C09080=1062.596,-86.701,-61.931,171.565,25.593,154.776
C09081=1062.602,-86.451,-61.943,171.566,25.594,154.776
C09082=1062.608,-86.202,-61.953,171.568,25.596,154.777
C09083=1062.614,-85.953,-61.964,171.570,25.597,154.777
C09084=1062.620,-85.702,-61.975,171.571,25.598,154.777
C09085=1062.627,-85.453,-61.985,171.573,25.600,154.777
C09086=1062.633,-85.204,-61.996,171.575,25.601,154.777
C09087=1062.639,-84.954,-62.007,171.576,25.603,154.777
C09088=1062.646,-84.704,-62.018,171.578,25.604,154.777
C09089=1062.652,-84.454,-62.028,171.580,25.605,154.777
C09090=1062.657,-84.204,-62.039,171.581,25.607,154.777
C09091=1062.664,-83.955,-62.049,171.583,25.608,154.777
C09092=1062.670,-83.705,-62.061,171.585,25.609,154.777
C09093=1062.676,-83.455,-62.072,171.587,25.611,154.777
C09094=1062.682,-83.206,-62.082,171.589,25.613,154.777
C09095=1062.689,-82.956,-62.093,171.591,25.614,154.777
C09096=1062.696,-82.674,-62.105,171.592,25.616,154.777
C09097=1062.703,-82.392,-62.118,171.594,25.617,154.778
C09098=1062.709,-82.110,-62.130,171.597,25.619,154.778
C09099=1062.716,-81.829,-62.143,171.598,25.621,154.778
C09100=1062.723,-81.579,-62.154,171.600,25.622,154.778
C09101=1062.729,-81.329,-62.164,171.602,25.624,154.778
C09102=1062.736,-81.079,-62.176,171.603,25.625,154.778
C09103=1062.741,-80.830,-62.187,171.605,25.627,154.778
C09104=1062.748,-80.580,-62.197,171.607,25.628,154.778
C09105=1062.754,-80.330,-62.208,171.608,25.630,154.778
C09106=1062.760,-80.081,-62.219,171.610,25.631,154.778
C09107=1062.766,-79.831,-62.230,171.612,25.632,154.778
C09108=1062.773,-79.582,-62.240,171.613,25.634,154.778
C09109=1062.779,-79.331,-62.252,171.615,25.635,154.778
C09110=1062.785,-79.082,-62.263,171.617,25.637,154.778
C09111=1062.791,-78.832,-62.274,171.619,25.639,154.779
C09112=1062.797,-78.583,-62.285,171.621,25.640,154.779
C09113=1062.803,-78.333,-62.296,171.622,25.642,154.779
C09114=1062.809,-78.083,-62.308,171.624,25.644,154.779
C09115=1062.815,-77.834,-62.318,171.626,25.645,154.779
C09116=1062.821,-77.583,-62.330,171.627,25.646,154.779
C09117=1062.827,-77.334,-62.341,171.629,25.648,154.779
C09118=1062.834,-77.084,-62.353,171.631,25.649,154.779
C09119=1062.839,-76.835,-62.363,171.632,25.651,154.779
C09120=1062.846,-76.585,-62.375,171.634,25.652,154.779
C09121=1062.851,-76.335,-62.386,171.636,25.654,154.779
C09122=1062.857,-76.086,-62.396,171.637,25.656,154.780
C09123=1062.864,-75.836,-62.408,171.639,25.657,154.780
C09124=1062.870,-75.587,-62.419,171.640,25.659,154.780
C09125=1062.877,-75.337,-62.430,171.642,25.661,154.780
C09126=1062.882,-75.087,-62.441,171.644,25.662,154.780
C09127=1062.889,-74.838,-62.453,171.645,25.664,154.780
C09128=1062.895,-74.588,-62.464,171.647,25.665,154.780
C09129=1062.901,-74.338,-62.475,171.650,25.667,154.780
C09130=1062.907,-74.089,-62.486,171.651,25.669,154.780
C09131=1062.914,-73.839,-62.498,171.653,25.671,154.780
C09132=1062.919,-73.589,-62.509,171.654,25.672,154.781
C09133=1062.925,-73.339,-62.520,171.656,25.673,154.781
C09134=1062.931,-73.090,-62.532,171.658,25.675,154.781
C09135=1062.937,-72.840,-62.543,171.659,25.677,154.781
C09136=1062.943,-72.590,-62.554,171.661,25.679,154.781
C09137=1062.950,-72.341,-62.566,171.663,25.681,154.781
C09138=1062.955,-72.091,-62.578,171.664,25.682,154.781
C09139=1062.960,-71.842,-62.588,171.666,25.684,154.781
C09140=1062.967,-71.592,-62.600,171.668,25.685,154.782
C09141=1062.973,-71.342,-62.611,171.669,25.687,154.782
C09142=1062.979,-71.092,-62.622,171.671,25.689,154.782
C09143=1062.984,-70.843,-62.635,171.672,25.691,154.782
C09144=1062.991,-70.593,-62.646,171.674,25.692,154.782
C09145=1062.997,-70.344,-62.658,171.676,25.694,154.782
C09146=1063.003,-70.094,-62.669,171.677,25.696,154.782
C09147=1063.008,-69.844,-62.680,171.679,25.698,154.783
C09148=1063.015,-69.594,-62.692,171.680,25.699,154.783
C09149=1063.021,-69.345,-62.703,171.682,25.701,154.783
C09150=1063.027,-69.095,-62.715,171.684,25.702,154.783
C09151=1063.034,-68.845,-62.726,171.686,25.705,154.783
C09152=1063.039,-68.596,-62.738,171.688,25.706,154.783
C09153=1063.045,-68.346,-62.750,171.689,25.708,154.783
C09154=1063.051,-68.096,-62.761,171.691,25.710,154.783
C09155=1063.058,-67.847,-62.773,171.693,25.712,154.783
C09156=1063.063,-67.597,-62.784,171.694,25.713,154.784
C09157=1063.069,-67.347,-62.796,171.696,25.715,154.784
C09158=1063.075,-67.098,-62.807,171.697,25.717,154.784
C09159=1063.082,-66.848,-62.819,171.699,25.719,154.784
C09160=1063.088,-66.569,-62.832,171.701,25.721,154.784
C09161=1063.095,-66.289,-62.845,171.702,25.722,154.784
C09162=1063.102,-66.009,-62.858,171.705,25.724,154.784
C09163=1063.108,-65.729,-62.871,171.706,25.726,154.785
C09164=1063.114,-65.480,-62.883,171.708,25.728,154.785
C09165=1063.121,-65.230,-62.895,171.710,25.730,154.785
C09166=1063.127,-64.981,-62.906,171.711,25.731,154.785
C09167=1063.132,-64.731,-62.918,171.713,25.733,154.785
C09168=1063.139,-64.481,-62.929,171.714,25.735,154.785
C09169=1063.145,-64.232,-62.941,171.716,25.737,154.785
C09170=1063.151,-63.982,-62.952,171.718,25.739,154.786
C09171=1063.157,-63.732,-62.965,171.719,25.740,154.786
C09172=1063.163,-63.483,-62.976,171.721,25.742,154.786
C09173=1063.169,-63.233,-62.988,171.723,25.744,154.786
C09174=1063.175,-62.984,-63.000,171.725,25.746,154.786
C09175=1063.181,-62.733,-63.011,171.726,25.748,154.786
C09176=1063.188,-62.484,-63.023,171.728,25.749,154.786
C09177=1063.194,-62.235,-63.035,171.730,25.751,154.786
C09178=1063.199,-61.984,-63.046,171.731,25.754,154.787
C09179=1063.206,-61.735,-63.058,171.733,25.755,154.787
C09180=1063.212,-61.486,-63.070,171.734,25.757,154.787
C09181=1063.218,-61.235,-63.082,171.736,25.759,154.787
C09182=1063.224,-60.986,-63.094,171.738,25.761,154.787
C09183=1063.230,-60.737,-63.105,171.739,25.762,154.787
C09184=1063.236,-60.486,-63.117,171.741,25.764,154.788
C09185=1063.243,-60.237,-63.129,171.742,25.766,154.788
C09186=1063.249,-59.987,-63.141,171.744,25.768,154.788
C09187=1063.255,-59.738,-63.153,171.746,25.769,154.788
C09188=1063.261,-59.488,-63.164,171.747,25.771,154.788
C09189=1063.268,-59.238,-63.176,171.749,25.773,154.788
C09190=1063.273,-58.989,-63.189,171.750,25.775,154.788
C09191=1063.280,-58.740,-63.201,171.752,25.777,154.789
C09192=1063.286,-58.489,-63.212,171.754,25.778,154.789
C09193=1063.292,-58.240,-63.224,171.755,25.780,154.789
C09194=1063.298,-57.991,-63.236,171.757,25.782,154.789
C09195=1063.304,-57.741,-63.248,171.758,25.784,154.789
C09196=1063.310,-57.491,-63.260,171.760,25.786,154.789
C09197=1063.317,-57.241,-63.272,171.762,25.788,154.790
C09198=1063.323,-56.992,-63.283,171.764,25.790,154.790
C09199=1063.329,-56.742,-63.296,171.766,25.792,154.790
C09200=1063.335,-56.493,-63.308,171.767,25.793,154.790
C09201=1063.342,-56.243,-63.319,171.769,25.795,154.790
C09202=1063.347,-55.993,-63.331,171.770,25.797,154.790
C09203=1063.354,-55.744,-63.343,171.772,25.799,154.791
C09204=1063.360,-55.494,-63.355,171.774,25.801,154.791
C09205=1063.366,-55.244,-63.368,171.775,25.803,154.791
C09206=1063.373,-54.995,-63.380,171.777,25.805,154.791
C09207=1063.378,-54.746,-63.392,171.778,25.806,154.791
C09208=1063.384,-54.495,-63.403,171.780,25.808,154.791
C09209=1063.391,-54.246,-63.415,171.781,25.810,154.791
C09210=1063.397,-53.996,-63.428,171.783,25.812,154.792
C09211=1063.404,-53.746,-63.440,171.785,25.814,154.792
C09212=1063.409,-53.497,-63.452,171.786,25.816,154.792
C09213=1063.416,-53.248,-63.464,171.788,25.817,154.792
C09214=1063.422,-52.998,-63.476,171.790,25.819,154.792
C09215=1063.428,-52.748,-63.488,171.791,25.822,154.792
C09216=1063.435,-52.499,-63.500,171.793,25.823,154.793
C09217=1063.441,-52.249,-63.513,171.794,25.825,154.793
C09218=1063.447,-51.999,-63.525,171.796,25.827,154.793
C09219=1063.453,-51.750,-63.536,171.797,25.829,154.793
C09220=1063.459,-51.500,-63.549,171.799,25.830,154.793
C09221=1063.466,-51.250,-63.560,171.801,25.833,154.793
C09222=1063.472,-51.000,-63.573,171.803,25.835,154.794
C09223=1063.478,-50.751,-63.585,171.805,25.837,154.794
C09224=1063.485,-50.473,-63.599,171.806,25.839,154.794
C09225=1063.492,-50.195,-63.612,171.808,25.841,154.794
C09226=1063.499,-49.916,-63.626,171.809,25.843,154.794
C09227=1063.506,-49.637,-63.640,171.812,25.845,154.794
C09228=1063.511,-49.387,-63.652,171.813,25.847,154.795
C09229=1063.518,-49.138,-63.664,171.815,25.849,154.795
C09230=1063.523,-48.889,-63.676,171.816,25.852,154.795
C09231=1063.529,-48.639,-63.689,171.818,25.853,154.795
C09232=1063.535,-48.389,-63.701,171.820,25.855,154.795
C09233=1063.542,-48.140,-63.714,171.821,25.857,154.796
C09234=1063.548,-47.890,-63.727,171.823,25.859,154.796
C09235=1063.554,-47.640,-63.739,171.824,25.862,154.796
C09236=1063.560,-47.391,-63.751,171.826,25.863,154.796
C09237=1063.566,-47.141,-63.763,171.827,25.866,154.796
C09238=1063.572,-46.891,-63.776,171.829,25.867,154.797
C09239=1063.578,-46.642,-63.788,171.830,25.870,154.797
C09240=1063.584,-46.392,-63.800,171.832,25.872,154.797
C09241=1063.591,-46.143,-63.814,171.834,25.873,154.797
C09242=1063.597,-45.893,-63.826,171.835,25.876,154.797
C09243=1063.602,-45.644,-63.838,171.837,25.877,154.798
C09244=1063.609,-45.394,-63.850,171.838,25.880,154.798
C09245=1063.614,-45.144,-63.863,171.840,25.881,154.798
C09246=1063.620,-44.894,-63.875,171.841,25.884,154.798
C09247=1063.627,-44.645,-63.888,171.843,25.886,154.798
C09248=1063.633,-44.396,-63.901,171.844,25.888,154.799
C09249=1063.639,-44.146,-63.913,171.846,25.890,154.799
C09250=1063.645,-43.896,-63.926,171.847,25.892,154.799
C09251=1063.652,-43.646,-63.938,171.849,25.894,154.799
C09252=1063.657,-43.398,-63.951,171.851,25.896,154.799
C09253=1063.663,-43.148,-63.963,171.852,25.898,154.800
C09254=1063.669,-42.898,-63.976,171.854,25.900,154.800
C09255=1063.675,-42.648,-63.988,171.855,25.902,154.800
C09256=1063.682,-42.399,-64.001,171.857,25.904,154.800
C09257=1063.688,-42.149,-64.013,171.858,25.906,154.800
C09258=1063.694,-41.899,-64.026,171.860,25.908,154.801
C09259=1063.700,-41.649,-64.039,171.862,25.910,154.801
C09260=1063.707,-41.400,-64.051,171.864,25.912,154.801
C09261=1063.713,-41.151,-64.064,171.865,25.915,154.801
C09262=1063.718,-40.901,-64.076,171.867,25.917,154.801
C09263=1063.725,-40.651,-64.090,171.869,25.919,154.802
C09264=1063.731,-40.402,-64.102,171.870,25.921,154.802
C09265=1063.737,-40.152,-64.114,171.872,25.923,154.802
C09266=1063.743,-39.903,-64.127,171.873,25.925,154.802
C09267=1063.749,-39.653,-64.140,171.875,25.927,154.802
C09268=1063.755,-39.403,-64.153,171.876,25.929,154.803
C09269=1063.761,-39.154,-64.166,171.878,25.931,154.803
C09270=1063.768,-38.904,-64.178,171.879,25.933,154.803
C09271=1063.774,-38.654,-64.190,171.881,25.935,154.803
C09272=1063.780,-38.405,-64.204,171.882,25.937,154.804
C09273=1063.786,-38.155,-64.216,171.884,25.940,154.804
C09274=1063.792,-37.906,-64.229,171.886,25.941,154.804
C09275=1063.798,-37.656,-64.242,171.887,25.944,154.804
C09276=1063.804,-37.406,-64.255,171.889,25.946,154.804
C09277=1063.810,-37.157,-64.268,171.890,25.948,154.805
C09278=1063.816,-36.907,-64.280,171.892,25.950,154.805
C09279=1063.823,-36.658,-64.294,171.893,25.953,154.805
C09280=1063.828,-36.408,-64.306,171.895,25.954,154.805
C09281=1063.835,-36.158,-64.319,171.896,25.957,154.806
C09282=1063.841,-35.909,-64.332,171.898,25.959,154.806
C09283=1063.847,-35.659,-64.345,171.899,25.961,154.806
C09284=1063.853,-35.409,-64.358,171.901,25.963,154.806
C09285=1063.859,-35.160,-64.371,171.902,25.965,154.807
C09286=1063.865,-34.910,-64.384,171.904,25.967,154.807
C09287=1063.871,-34.661,-64.397,171.905,25.970,154.807
C09288=1063.877,-34.382,-64.411,171.907,25.972,154.807
C09289=1063.884,-34.105,-64.425,171.908,25.974,154.807
C09290=1063.891,-33.827,-64.439,171.911,25.977,154.808
C09291=1063.897,-33.548,-64.454,171.912,25.979,154.808
C09292=1063.904,-33.299,-64.468,171.914,25.981,154.808
C09293=1063.910,-33.049,-64.480,171.915,25.984,154.808
C09294=1063.916,-32.800,-64.494,171.917,25.986,154.809
C09295=1063.922,-32.551,-64.507,171.918,25.988,154.809
C09296=1063.928,-32.301,-64.519,171.920,25.990,154.809
C09297=1063.934,-32.051,-64.533,171.921,25.993,154.809
C09298=1063.940,-31.801,-64.545,171.923,25.994,154.810
C09299=1063.946,-31.552,-64.558,171.924,25.997,154.810
C09300=1063.952,-31.303,-64.572,171.926,25.999,154.810
C09301=1063.958,-31.053,-64.584,171.927,26.001,154.810
C09302=1063.965,-30.804,-64.598,171.929,26.003,154.811
C09303=1063.971,-30.554,-64.610,171.931,26.005,154.811
C09304=1063.977,-30.304,-64.624,171.932,26.008,154.811
C09305=1063.984,-30.055,-64.637,171.934,26.010,154.811
C09306=1063.989,-29.805,-64.650,171.935,26.012,154.811
C09307=1063.995,-29.555,-64.663,171.937,26.014,154.812
C09308=1064.001,-29.306,-64.677,171.938,26.016,154.812
C09309=1064.007,-29.056,-64.689,171.940,26.019,154.812
C09310=1064.013,-28.807,-64.702,171.941,26.021,154.812
C09311=1064.019,-28.558,-64.716,171.943,26.023,154.813
C09312=1064.026,-28.307,-64.729,171.944,26.025,154.813
C09313=1064.032,-28.058,-64.742,171.946,26.028,154.813
C09314=1064.038,-27.808,-64.755,171.947,26.029,154.813
C09315=1064.045,-27.559,-64.768,171.949,26.032,154.814
C09316=1064.051,-27.309,-64.781,171.950,26.034,154.814
C09317=1064.056,-27.060,-64.795,171.952,26.036,154.814
C09318=1064.063,-26.810,-64.809,171.953,26.039,154.814
C09319=1064.069,-26.561,-64.822,171.955,26.040,154.815
C09320=1064.075,-26.311,-64.834,171.956,26.043,154.815
C09321=1064.080,-26.061,-64.848,171.958,26.045,154.815
C09322=1064.087,-25.812,-64.861,171.959,26.047,154.815
C09323=1064.093,-25.563,-64.875,171.961,26.050,154.816
C09324=1064.099,-25.313,-64.887,171.962,26.052,154.816
C09325=1064.104,-25.063,-64.901,171.964,26.054,154.816
C09326=1064.111,-24.813,-64.915,171.965,26.057,154.816
C09327=1064.117,-24.564,-64.928,171.967,26.059,154.817
C09328=1064.123,-24.314,-64.942,171.968,26.061,154.817
C09329=1064.129,-24.065,-64.955,171.970,26.064,154.817
C09330=1064.135,-23.815,-64.968,171.971,26.066,154.817
C09331=1064.140,-23.566,-64.982,171.973,26.068,154.818
C09332=1064.147,-23.316,-64.995,171.975,26.070,154.818
C09333=1064.153,-23.066,-65.009,171.976,26.072,154.818
C09334=1064.159,-22.817,-65.022,171.978,26.075,154.818
C09335=1064.165,-22.567,-65.036,171.979,26.077,154.819
C09336=1064.171,-22.318,-65.049,171.981,26.079,154.819
C09337=1064.177,-22.069,-65.063,171.982,26.082,154.819
C09338=1064.183,-21.818,-65.076,171.984,26.084,154.820
C09339=1064.189,-21.569,-65.089,171.985,26.086,154.820
C09340=1064.195,-21.319,-65.103,171.987,26.089,154.820
C09341=1064.201,-21.070,-65.116,171.988,26.091,154.820
C09342=1064.207,-20.821,-65.129,171.990,26.093,154.821
C09343=1064.213,-20.570,-65.144,171.991,26.096,154.821
C09344=1064.220,-20.321,-65.157,171.993,26.098,154.821
C09345=1064.226,-20.072,-65.170,171.994,26.100,154.821
C09346=1064.231,-19.822,-65.184,171.996,26.103,154.822
C09347=1064.238,-19.572,-65.198,171.997,26.105,154.822
C09348=1064.244,-19.323,-65.211,171.999,26.107,154.822
C09349=1064.250,-19.074,-65.225,172.000,26.110,154.822
C09350=1064.256,-18.824,-65.238,172.002,26.112,154.823
C09351=1064.263,-18.574,-65.252,172.003,26.114,154.823
C09352=1064.269,-18.295,-65.267,172.005,26.117,154.823
C09353=1064.276,-18.016,-65.283,172.006,26.119,154.824
C09354=1064.282,-17.738,-65.298,172.008,26.122,154.824
C09355=1064.289,-17.459,-65.313,172.010,26.124,154.824
C09356=1064.295,-17.210,-65.326,172.011,26.127,154.824
C09357=1064.302,-16.960,-65.340,172.013,26.129,154.825
C09358=1064.308,-16.710,-65.354,172.014,26.131,154.825
C09359=1064.314,-16.461,-65.367,172.016,26.134,154.825
C09360=1064.320,-16.211,-65.381,172.017,26.136,154.825
C09361=1064.326,-15.961,-65.394,172.019,26.138,154.826
C09362=1064.333,-15.713,-65.408,172.020,26.141,154.826
C09363=1064.338,-15.463,-65.422,172.022,26.143,154.826
C09364=1064.345,-15.213,-65.436,172.023,26.145,154.827
C09365=1064.351,-14.964,-65.450,172.025,26.148,154.827
C09366=1064.357,-14.714,-65.463,172.026,26.150,154.827
C09367=1064.363,-14.464,-65.477,172.028,26.152,154.827
C09368=1064.369,-14.215,-65.490,172.029,26.155,154.828
C09369=1064.375,-13.965,-65.504,172.031,26.157,154.828
C09370=1064.380,-13.716,-65.519,172.032,26.159,154.828
C09371=1064.387,-13.466,-65.533,172.034,26.162,154.829
C09372=1064.393,-13.217,-65.546,172.035,26.164,154.829
C09373=1064.399,-12.967,-65.560,172.037,26.167,154.829
C09374=1064.405,-12.717,-65.574,172.038,26.169,154.829
C09375=1064.411,-12.468,-65.588,172.040,26.171,154.830
C09376=1064.417,-12.219,-65.602,172.041,26.174,154.830
C09377=1064.423,-11.969,-65.616,172.043,26.176,154.830
C09378=1064.429,-11.719,-65.629,172.043,26.178,154.830
C09379=1064.435,-11.470,-65.643,172.045,26.181,154.831
C09380=1064.441,-11.220,-65.658,172.046,26.183,154.831
C09381=1064.447,-10.971,-65.671,172.048,26.186,154.831
C09382=1064.453,-10.721,-65.685,172.049,26.188,154.832
C09383=1064.459,-10.471,-65.699,172.051,26.190,154.832
C09384=1064.465,-10.222,-65.713,172.052,26.192,154.832
C09385=1064.471,-9.973,-65.727,172.054,26.195,154.832
C09386=1064.478,-9.723,-65.741,172.055,26.198,154.833
C09387=1064.483,-9.474,-65.756,172.057,26.200,154.833
C09388=1064.489,-9.224,-65.769,172.058,26.202,154.833
C09389=1064.496,-8.974,-65.783,172.060,26.205,154.834
C09390=1064.501,-8.725,-65.798,172.061,26.207,154.834
C09391=1064.508,-8.475,-65.812,172.063,26.209,154.834
C09392=1064.514,-8.226,-65.825,172.064,26.212,154.835
C09393=1064.520,-7.977,-65.840,172.066,26.214,154.835
C09394=1064.526,-7.727,-65.854,172.067,26.217,154.835
C09395=1064.532,-7.477,-65.867,172.069,26.219,154.835
C09396=1064.538,-7.228,-65.882,172.070,26.221,154.836
C09397=1064.544,-6.978,-65.896,172.072,26.224,154.836
C09398=1064.550,-6.729,-65.909,172.073,26.227,154.836
C09399=1064.556,-6.479,-65.924,172.075,26.229,154.837
C09400=1064.562,-6.230,-65.938,172.076,26.231,154.837
C09401=1064.569,-5.980,-65.952,172.078,26.234,154.837
C09402=1064.574,-5.731,-65.966,172.079,26.236,154.837
C09403=1064.580,-5.480,-65.980,172.081,26.238,154.838
C09404=1064.587,-5.232,-65.994,172.082,26.241,154.838
C09405=1064.592,-4.982,-66.008,172.084,26.243,154.838
C09406=1064.599,-4.733,-66.023,172.085,26.246,154.839
C09407=1064.605,-4.483,-66.037,172.087,26.248,154.839
C09408=1064.611,-4.234,-66.052,172.088,26.250,154.839
C09409=1064.617,-3.984,-66.065,172.090,26.253,154.839
C09410=1064.623,-3.734,-66.080,172.091,26.256,154.840
C09411=1064.630,-3.485,-66.094,172.092,26.258,154.840
C09412=1064.636,-3.235,-66.108,172.094,26.260,154.840
C09413=1064.641,-2.986,-66.122,172.095,26.262,154.841
C09414=1064.647,-2.736,-66.137,172.097,26.265,154.841
C09415=1064.653,-2.487,-66.151,172.097,26.267,154.841
C09416=1064.660,-2.206,-66.168,172.100,26.271,154.842
C09417=1064.667,-1.926,-66.183,172.101,26.273,154.842
C09418=1064.674,-1.645,-66.199,172.103,26.276,154.842
C09419=1064.680,-1.365,-66.216,172.104,26.279,154.843
C09420=1064.685,-1.116,-66.230,172.106,26.281,154.843
C09421=1064.692,-0.866,-66.245,172.107,26.284,154.843
C09422=1064.697,-0.616,-66.259,172.108,26.286,154.844
C09423=1064.704,-0.367,-66.274,172.110,26.288,154.844
C09424=1064.709,-0.117,-66.288,172.111,26.291,154.844
C09425=1064.716,0.132,-66.302,172.113,26.294,154.845
C09426=1064.722,0.381,-66.317,172.114,26.296,154.845
C09427=1064.728,0.631,-66.331,172.116,26.299,154.845
C09428=1064.734,0.880,-66.345,172.117,26.301,154.845
C09429=1064.740,1.130,-66.360,172.119,26.304,154.846
C09430=1064.746,1.380,-66.374,172.120,26.306,154.846
C09431=1064.752,1.629,-66.389,172.122,26.309,154.846
C09432=1064.758,1.878,-66.404,172.123,26.312,154.847
C09433=1064.764,2.128,-66.418,172.125,26.314,154.847
C09434=1064.770,2.377,-66.433,172.126,26.316,154.847
C09435=1064.776,2.627,-66.447,172.128,26.319,154.848
C09436=1064.782,2.877,-66.461,172.129,26.321,154.848
C09437=1064.788,3.126,-66.476,172.131,26.324,154.848
C09438=1064.794,3.375,-66.491,172.131,26.326,154.849
C09439=1064.800,3.625,-66.505,172.133,26.329,154.849
C09440=1064.806,3.874,-66.520,172.134,26.331,154.849
C09441=1064.812,4.124,-66.535,172.136,26.334,154.850
C09442=1064.818,4.373,-66.549,172.137,26.336,154.850
C09443=1064.824,4.623,-66.563,172.138,26.339,154.850
C09444=1064.830,4.872,-66.578,172.140,26.341,154.851
C09445=1064.836,5.122,-66.593,172.141,26.344,154.851
C09446=1064.842,5.371,-66.608,172.143,26.346,154.851
C09447=1064.847,5.621,-66.622,172.144,26.349,154.852
C09448=1064.854,5.871,-66.637,172.146,26.351,154.852
C09449=1064.859,6.120,-66.652,172.147,26.354,154.852
C09450=1064.866,6.370,-66.667,172.149,26.356,154.852
C09451=1064.871,6.619,-66.681,172.150,26.359,154.853
C09452=1064.878,6.869,-66.696,172.152,26.361,154.853
C09453=1064.883,7.118,-66.710,172.153,26.364,154.853
C09454=1064.890,7.368,-66.725,172.155,26.367,154.854
C09455=1064.896,7.617,-66.740,172.156,26.369,154.854
C09456=1064.902,7.866,-66.755,172.158,26.371,154.854
C09457=1064.908,8.116,-66.769,172.159,26.374,154.855
C09458=1064.914,8.365,-66.784,172.161,26.376,154.855
C09459=1064.920,8.615,-66.798,172.162,26.379,154.855
C09460=1064.927,8.865,-66.813,172.163,26.381,154.856
C09461=1064.932,9.114,-66.828,172.164,26.384,154.856
C09462=1064.939,9.363,-66.843,172.166,26.386,154.856
C09463=1064.945,9.613,-66.858,172.167,26.389,154.857
C09464=1064.951,9.862,-66.872,172.169,26.391,154.857
C09465=1064.957,10.112,-66.887,172.170,26.394,154.857
C09466=1064.963,10.362,-66.902,172.172,26.396,154.858
C09467=1064.968,10.611,-66.917,172.173,26.399,154.858
C09468=1064.975,10.861,-66.932,172.174,26.401,154.858
C09469=1064.981,11.110,-66.947,172.176,26.404,154.858
C09470=1064.987,11.359,-66.961,172.177,26.407,154.859
C09471=1064.993,11.609,-66.976,172.179,26.409,154.859
C09472=1065.000,11.859,-66.991,172.180,26.411,154.859
C09473=1065.005,12.108,-67.006,172.182,26.414,154.860
C09474=1065.012,12.357,-67.021,172.183,26.416,154.860
C09475=1065.018,12.607,-67.036,172.185,26.419,154.860
C09476=1065.024,12.856,-67.050,172.186,26.422,154.861
C09477=1065.030,13.106,-67.066,172.188,26.424,154.861
C09478=1065.036,13.356,-67.081,172.189,26.427,154.861
C09479=1065.042,13.605,-67.096,172.191,26.429,154.862
C09480=1065.049,13.887,-67.112,172.192,26.432,154.862
C09481=1065.056,14.170,-67.129,172.194,26.435,154.862
C09482=1065.063,14.452,-67.146,172.195,26.437,154.863
C09483=1065.070,14.735,-67.163,172.196,26.440,154.863
C09484=1065.075,14.984,-67.178,172.198,26.443,154.864
C09485=1065.082,15.233,-67.193,172.199,26.445,154.864
C09486=1065.088,15.483,-67.208,172.201,26.448,154.864
C09487=1065.093,15.732,-67.224,172.202,26.450,154.864
C09488=1065.100,15.981,-67.239,172.204,26.453,154.865
C09489=1065.106,16.231,-67.254,172.205,26.456,154.865
C09490=1065.112,16.481,-67.269,172.207,26.458,154.866
C09491=1065.118,16.730,-67.284,172.208,26.461,154.866
C09492=1065.124,16.980,-67.299,172.210,26.464,154.866
C09493=1065.130,17.230,-67.314,172.211,26.466,154.866
C09494=1065.135,17.479,-67.329,172.213,26.469,154.867
C09495=1065.142,17.728,-67.345,172.214,26.471,154.867
C09496=1065.148,17.978,-67.360,172.215,26.474,154.867
C09497=1065.154,18.227,-67.375,172.217,26.476,154.868
C09498=1065.160,18.476,-67.390,172.217,26.479,154.868
C09499=1065.165,18.726,-67.405,172.219,26.481,154.868
C09500=1065.172,18.976,-67.420,172.220,26.484,154.869
C09501=1065.179,19.225,-67.436,172.222,26.486,154.869
C09502=1065.184,19.474,-67.451,172.223,26.489,154.870
C09503=1065.190,19.724,-67.466,172.225,26.491,154.870
C09504=1065.196,19.973,-67.481,172.226,26.494,154.870
C09505=1065.202,20.223,-67.497,172.228,26.497,154.870
C09506=1065.208,20.472,-67.512,172.229,26.499,154.871
C09507=1065.214,20.722,-67.527,172.231,26.502,154.871
C09508=1065.220,20.971,-67.542,172.232,26.505,154.872
C09509=1065.227,21.220,-67.558,172.234,26.507,154.872
C09510=1065.232,21.470,-67.573,172.235,26.510,154.872
C09511=1065.238,21.719,-67.588,172.237,26.513,154.873
C09512=1065.244,21.969,-67.603,172.238,26.515,154.873
C09513=1065.251,22.218,-67.619,172.240,26.518,154.873
C09514=1065.256,22.468,-67.634,172.240,26.520,154.874
C09515=1065.262,22.717,-67.649,172.242,26.523,154.874
C09516=1065.268,22.967,-67.666,172.243,26.526,154.874
C09517=1065.274,23.216,-67.680,172.244,26.528,154.875
C09518=1065.280,23.466,-67.696,172.246,26.531,154.875
C09519=1065.286,23.715,-67.711,172.247,26.533,154.875
C09520=1065.292,23.965,-67.727,172.249,26.536,154.876
C09521=1065.298,24.214,-67.742,172.250,26.538,154.876
C09522=1065.304,24.464,-67.758,172.252,26.541,154.876
C09523=1065.310,24.713,-67.773,172.253,26.544,154.877
C09524=1065.316,24.962,-67.789,172.255,26.546,154.877
C09525=1065.322,25.211,-67.804,172.256,26.549,154.877
C09526=1065.328,25.461,-67.819,172.258,26.551,154.878
C09527=1065.334,25.710,-67.835,172.259,26.554,154.878
C09528=1065.340,25.960,-67.851,172.261,26.556,154.878
C09529=1065.347,26.210,-67.866,172.262,26.559,154.879
C09530=1065.352,26.459,-67.881,172.263,26.561,154.879
C09531=1065.358,26.708,-67.896,172.264,26.564,154.879
C09532=1065.364,26.958,-67.913,172.265,26.567,154.880
C09533=1065.371,27.207,-67.928,172.267,26.569,154.880
C09534=1065.377,27.457,-67.944,172.268,26.572,154.881
C09535=1065.382,27.707,-67.959,172.270,26.575,154.881
C09536=1065.389,27.956,-67.975,172.271,26.577,154.881
C09537=1065.394,28.205,-67.990,172.273,26.580,154.882
C09538=1065.401,28.454,-68.006,172.274,26.583,154.882
C09539=1065.406,28.704,-68.021,172.276,26.585,154.882
C09540=1065.412,28.953,-68.038,172.277,26.588,154.883
C09541=1065.419,29.203,-68.053,172.279,26.591,154.883
C09542=1065.425,29.452,-68.069,172.280,26.593,154.883
C09543=1065.430,29.702,-68.084,172.282,26.596,154.884
C09544=1065.437,29.986,-68.102,172.283,26.599,154.884
C09545=1065.444,30.269,-68.120,172.284,26.602,154.884
C09546=1065.451,30.553,-68.138,172.286,26.605,154.885
C09547=1065.457,30.837,-68.156,172.287,26.608,154.885
C09548=1065.464,31.086,-68.171,172.289,26.611,154.886
C09549=1065.469,31.335,-68.187,172.290,26.613,154.886
C09550=1065.475,31.585,-68.203,172.292,26.616,154.886
C09551=1065.481,31.834,-68.218,172.293,26.618,154.887
C09552=1065.487,32.083,-68.235,172.295,26.621,154.887
C09553=1065.493,32.333,-68.250,172.296,26.624,154.887
C09554=1065.499,32.583,-68.266,172.298,26.626,154.888
C09555=1065.506,32.832,-68.282,172.299,26.629,154.888
C09556=1065.511,33.082,-68.298,172.300,26.632,154.888
C09557=1065.517,33.331,-68.314,172.302,26.634,154.889
C09558=1065.523,33.580,-68.330,172.303,26.637,154.889
C09559=1065.529,33.830,-68.345,172.305,26.640,154.890
C09560=1065.535,34.079,-68.361,172.306,26.642,154.890
C09561=1065.541,34.328,-68.377,172.308,26.645,154.890
C09562=1065.546,34.578,-68.393,172.308,26.647,154.891
C09563=1065.553,34.827,-68.408,172.310,26.650,154.891
C09564=1065.559,35.076,-68.425,172.311,26.653,154.891
C09565=1065.565,35.326,-68.440,172.313,26.655,154.892
C09566=1065.571,35.576,-68.457,172.314,26.658,154.892
C09567=1065.577,35.825,-68.472,172.316,26.661,154.892
C09568=1065.583,36.074,-68.488,172.317,26.663,154.893
C09569=1065.589,36.324,-68.504,172.319,26.666,154.893
C09570=1065.595,36.573,-68.520,172.320,26.669,154.893
C09571=1065.602,36.823,-68.536,172.322,26.671,154.894
C09572=1065.608,37.072,-68.552,172.323,26.674,154.894
C09573=1065.613,37.322,-68.568,172.325,26.676,154.894
C09574=1065.619,37.571,-68.584,172.326,26.679,154.895
C09575=1065.625,37.821,-68.600,172.327,26.682,154.895
C09576=1065.631,38.070,-68.616,172.329,26.684,154.895
C09577=1065.638,38.319,-68.632,172.329,26.687,154.896
C09578=1065.643,38.569,-68.648,172.331,26.689,154.896
C09579=1065.649,38.818,-68.664,172.332,26.692,154.897
C09580=1065.655,39.068,-68.680,172.334,26.695,154.897
C09581=1065.661,39.317,-68.696,172.335,26.697,154.897
C09582=1065.667,39.566,-68.713,172.337,26.700,154.898
C09583=1065.673,39.816,-68.729,172.338,26.703,154.898
C09584=1065.679,40.066,-68.744,172.340,26.705,154.898
C09585=1065.685,40.315,-68.761,172.341,26.708,154.899
C09586=1065.691,40.564,-68.777,172.343,26.711,154.899
C09587=1065.697,40.814,-68.793,172.344,26.713,154.899
C09588=1065.703,41.063,-68.810,172.346,26.716,154.900
C09589=1065.708,41.312,-68.826,172.347,26.719,154.900
C09590=1065.714,41.562,-68.842,172.348,26.722,154.901
C09591=1065.720,41.811,-68.858,172.350,26.724,154.901
C09592=1065.726,42.060,-68.875,172.350,26.727,154.901
C09593=1065.732,42.310,-68.891,172.352,26.730,154.902
C09594=1065.738,42.559,-68.907,172.353,26.732,154.902
C09595=1065.744,42.808,-68.923,172.355,26.735,154.902
C09596=1065.750,43.058,-68.939,172.356,26.738,154.903
C09597=1065.756,43.308,-68.955,172.358,26.740,154.903
C09598=1065.762,43.557,-68.971,172.359,26.743,154.903
C09599=1065.768,43.806,-68.988,172.361,26.746,154.904
C09600=1065.774,44.056,-69.004,172.362,26.748,154.904
C09601=1065.780,44.305,-69.020,172.364,26.751,154.905
C09602=1065.785,44.555,-69.037,172.365,26.754,154.905
C09603=1065.791,44.804,-69.054,172.367,26.756,154.905
C09604=1065.797,45.053,-69.070,172.368,26.759,154.906
C09605=1065.803,45.302,-69.086,172.369,26.762,154.906
C09606=1065.809,45.552,-69.103,172.371,26.765,154.906
C09607=1065.814,45.801,-69.120,172.371,26.768,154.907
C09608=1065.821,46.085,-69.138,172.374,26.771,154.907
C09609=1065.828,46.369,-69.157,172.375,26.774,154.908
C09610=1065.835,46.653,-69.176,172.377,26.777,154.908
C09611=1065.841,46.936,-69.194,172.378,26.780,154.909
C09612=1065.847,47.186,-69.210,172.379,26.783,154.909
C09613=1065.853,47.434,-69.227,172.381,26.785,154.909
C09614=1065.859,47.684,-69.243,172.382,26.788,154.910
C09615=1065.865,47.934,-69.261,172.384,26.791,154.910
C09616=1065.871,48.183,-69.277,172.385,26.793,154.910
C09617=1065.876,48.433,-69.293,172.387,26.796,154.911
C09618=1065.882,48.682,-69.309,172.388,26.799,154.911
C09619=1065.888,48.932,-69.326,172.390,26.801,154.912
C09620=1065.894,49.181,-69.343,172.391,26.804,154.912
C09621=1065.900,49.430,-69.359,172.393,26.807,154.912
C09622=1065.906,49.679,-69.376,172.394,26.810,154.913
C09623=1065.912,49.929,-69.392,172.395,26.812,154.913
C09624=1065.917,50.178,-69.409,172.396,26.815,154.913
C09625=1065.923,50.427,-69.426,172.398,26.818,154.914
C09626=1065.930,50.677,-69.442,172.399,26.820,154.914
C09627=1065.935,50.927,-69.459,172.400,26.823,154.915
C09628=1065.941,51.176,-69.475,172.402,26.826,154.915
C09629=1065.947,51.425,-69.492,172.403,26.828,154.915
C09630=1065.953,51.674,-69.509,172.405,26.831,154.916
C09631=1065.958,51.924,-69.526,172.406,26.834,154.916
C09632=1065.964,52.173,-69.542,172.408,26.837,154.916
C09633=1065.971,52.423,-69.558,172.409,26.839,154.917
C09634=1065.977,52.672,-69.575,172.411,26.842,154.917
C09635=1065.982,52.922,-69.592,172.412,26.845,154.918
C09636=1065.988,53.171,-69.608,172.414,26.848,154.918
C09637=1065.995,53.420,-69.625,172.415,26.850,154.918
C09638=1066.000,53.669,-69.642,172.416,26.853,154.919
C09639=1066.006,53.919,-69.659,172.417,26.855,154.919
C09640=1066.013,54.168,-69.676,172.419,26.858,154.919
C09641=1066.019,54.417,-69.692,172.420,26.861,154.920
C09642=1066.024,54.667,-69.709,172.422,26.863,154.920
C09643=1066.030,54.916,-69.726,172.423,26.866,154.921
C09644=1066.036,55.165,-69.742,172.424,26.869,154.921
C09645=1066.042,55.416,-69.759,172.426,26.872,154.921
C09646=1066.048,55.664,-69.776,172.427,26.874,154.922
C09647=1066.054,55.914,-69.793,172.429,26.877,154.922
C09648=1066.059,56.163,-69.810,172.430,26.880,154.922
C09649=1066.066,56.413,-69.827,172.432,26.883,154.923
C09650=1066.072,56.662,-69.843,172.433,26.885,154.923
C09651=1066.078,56.911,-69.860,172.435,26.888,154.923
C09652=1066.083,57.160,-69.877,172.436,26.891,154.924
C09653=1066.090,57.411,-69.894,172.438,26.893,154.924
C09654=1066.096,57.659,-69.911,172.439,26.896,154.925
C09655=1066.101,57.909,-69.927,172.440,26.898,154.925
C09656=1066.108,58.158,-69.944,172.441,26.901,154.925
C09657=1066.114,58.408,-69.961,172.443,26.903,154.926
C09658=1066.120,58.657,-69.979,172.444,26.906,154.926
C09659=1066.126,58.906,-69.995,172.446,26.909,154.926
C09660=1066.132,59.155,-70.012,172.447,26.912,154.927
C09661=1066.138,59.405,-70.029,172.449,26.914,154.927
C09662=1066.144,59.654,-70.046,172.450,26.917,154.927
C09663=1066.150,59.903,-70.062,172.452,26.920,154.928
C09664=1066.156,60.153,-70.080,172.453,26.923,154.928
C09665=1066.162,60.402,-70.096,172.455,26.925,154.929
C09666=1066.168,60.651,-70.114,172.456,26.928,154.929
C09667=1066.174,60.901,-70.130,172.458,26.931,154.929
C09668=1066.180,61.150,-70.148,172.459,26.933,154.930
C09669=1066.186,61.400,-70.164,172.461,26.936,154.930
C09670=1066.192,61.649,-70.181,172.462,26.939,154.930
C09671=1066.198,61.899,-70.198,172.463,26.941,154.931
C09672=1066.206,62.182,-70.218,172.465,26.944,154.931
C09673=1066.212,62.465,-70.237,172.466,26.947,154.932
C09674=1066.219,62.749,-70.257,172.468,26.950,154.932
C09675=1066.226,63.032,-70.276,172.470,26.953,154.932
C09676=1066.232,63.281,-70.293,172.471,26.956,154.933
C09677=1066.237,63.531,-70.310,172.472,26.958,154.933
C09678=1066.244,63.780,-70.327,172.474,26.961,154.933
C09679=1066.250,64.030,-70.344,172.475,26.964,154.934
C09680=1066.256,64.278,-70.361,172.477,26.966,154.934
C09681=1066.262,64.528,-70.379,172.478,26.969,154.935
C09682=1066.268,64.777,-70.395,172.480,26.971,154.935
C09683=1066.273,65.027,-70.413,172.481,26.974,154.935
C09684=1066.280,65.276,-70.430,172.483,26.977,154.936
C09685=1066.285,65.526,-70.447,172.484,26.980,154.936
C09686=1066.291,65.775,-70.465,172.485,26.983,154.937
C09687=1066.298,66.024,-70.482,172.487,26.986,154.937
C09688=1066.303,66.273,-70.499,172.489,26.988,154.937
C09689=1066.309,66.522,-70.516,172.490,26.991,154.938
C09690=1066.315,66.772,-70.534,172.491,26.994,154.938
C09691=1066.321,67.021,-70.551,172.493,26.996,154.938
C09692=1066.328,67.271,-70.568,172.494,26.999,154.939
C09693=1066.333,67.520,-70.585,172.496,27.001,154.939
C09694=1066.339,67.769,-70.603,172.497,27.004,154.939
C09695=1066.345,68.019,-70.620,172.499,27.007,154.940
C09696=1066.351,68.268,-70.638,172.500,27.010,154.940
C09697=1066.356,68.518,-70.655,172.501,27.012,154.941
C09698=1066.363,68.767,-70.672,172.502,27.015,154.941
C09699=1066.369,69.016,-70.690,172.504,27.018,154.941
C09700=1066.375,69.266,-70.708,172.505,27.020,154.942
C09701=1066.381,69.514,-70.725,172.507,27.023,154.942
C09702=1066.386,69.764,-70.741,172.508,27.026,154.943
C09703=1066.392,70.014,-70.759,172.510,27.028,154.943
C09704=1066.398,70.263,-70.776,172.511,27.031,154.943
C09705=1066.404,70.512,-70.794,172.513,27.034,154.944
C09706=1066.410,70.761,-70.812,172.514,27.037,154.944
C09707=1066.416,71.010,-70.829,172.516,27.040,154.944
C09708=1066.422,71.260,-70.847,172.517,27.042,154.945
C09709=1066.428,71.510,-70.864,172.519,27.045,154.945
C09710=1066.433,71.759,-70.881,172.520,27.048,154.946
C09711=1066.439,72.008,-70.899,172.522,27.050,154.946
C09712=1066.445,72.257,-70.917,172.523,27.053,154.946
C09713=1066.452,72.507,-70.934,172.525,27.056,154.947
C09714=1066.457,72.756,-70.952,172.526,27.059,154.947
C09715=1066.463,73.005,-70.969,172.527,27.062,154.948
C09716=1066.469,73.255,-70.987,172.529,27.064,154.948
C09717=1066.474,73.504,-71.005,172.530,27.067,154.948
C09718=1066.481,73.753,-71.023,172.532,27.070,154.949
C09719=1066.487,74.002,-71.040,172.533,27.072,154.949
C09720=1066.493,74.252,-71.057,172.534,27.075,154.949
C09721=1066.498,74.501,-71.075,172.535,27.078,154.950
C09722=1066.504,74.750,-71.093,172.537,27.080,154.950
C09723=1066.510,75.000,-71.111,172.538,27.083,154.951
C09724=1066.516,75.249,-71.128,172.540,27.086,154.951
C09725=1066.522,75.498,-71.145,172.541,27.088,154.951
C09726=1066.528,75.747,-71.163,172.543,27.091,154.952
C09727=1066.534,75.997,-71.181,172.544,27.094,154.952
C09728=1066.540,76.246,-71.198,172.546,27.096,154.952
C09729=1066.546,76.496,-71.216,172.547,27.099,154.953
C09730=1066.551,76.745,-71.234,172.549,27.102,154.953
C09731=1066.557,76.994,-71.252,172.550,27.105,154.954
C09732=1066.563,77.244,-71.269,172.552,27.108,154.954
C09733=1066.570,77.493,-71.287,172.553,27.110,154.954
C09734=1066.575,77.742,-71.304,172.555,27.113,154.955
C09735=1066.582,77.991,-71.323,172.556,27.116,154.955
C09736=1066.588,78.275,-71.343,172.558,27.118,154.955
C09737=1066.595,78.558,-71.363,172.559,27.122,154.956
C09738=1066.601,78.841,-71.384,172.562,27.125,154.956
C09739=1066.608,79.124,-71.404,172.563,27.128,154.957
C09740=1066.613,79.373,-71.422,172.564,27.131,154.957
C09741=1066.619,79.623,-71.440,172.566,27.133,154.958
C09742=1066.625,79.872,-71.457,172.567,27.136,154.958
C09743=1066.631,80.122,-71.475,172.569,27.139,154.958
C09744=1066.636,80.371,-71.493,172.570,27.142,154.959
C09745=1066.643,80.620,-71.512,172.572,27.145,154.959
C09746=1066.648,80.869,-71.529,172.573,27.147,154.960
C09747=1066.654,81.119,-71.547,172.575,27.150,154.960
C09748=1066.660,81.368,-71.565,172.576,27.153,154.960
C09749=1066.666,81.617,-71.583,172.578,27.155,154.961
C09750=1066.672,81.866,-71.601,172.579,27.158,154.961
C09751=1066.677,82.116,-71.619,172.581,27.161,154.961
C09752=1066.683,82.365,-71.637,172.582,27.164,154.962
C09753=1066.689,82.614,-71.656,172.584,27.167,154.962
C09754=1066.695,82.864,-71.674,172.584,27.169,154.963
C09755=1066.701,83.113,-71.691,172.586,27.172,154.963
C09756=1066.707,83.363,-71.709,172.587,27.175,154.963
C09757=1066.713,83.611,-71.727,172.589,27.177,154.964
C09758=1066.719,83.861,-71.745,172.590,27.180,154.964
C09759=1066.724,84.110,-71.763,172.592,27.183,154.965
C09760=1066.730,84.359,-71.782,172.593,27.185,154.965
C09761=1066.736,84.609,-71.800,172.595,27.188,154.965
C09762=1066.742,84.858,-71.818,172.596,27.191,154.966
C09763=1066.748,85.107,-71.836,172.598,27.194,154.966
C09764=1066.754,85.356,-71.854,172.599,27.196,154.966
C09765=1066.760,85.606,-71.872,172.601,27.199,154.967
C09766=1066.766,85.855,-71.890,172.602,27.202,154.967
C09767=1066.772,86.104,-71.908,172.604,27.205,154.968
C09768=1066.777,86.354,-71.926,172.605,27.207,154.968
C09769=1066.783,86.603,-71.945,172.607,27.210,154.968
C09770=1066.789,86.853,-71.963,172.608,27.212,154.969
C09771=1066.795,87.101,-71.981,172.610,27.215,154.969
C09772=1066.801,87.351,-71.999,172.611,27.218,154.970
C09773=1066.807,87.600,-72.017,172.613,27.221,154.970
C09774=1066.813,87.849,-72.035,172.614,27.224,154.970
C09775=1066.818,88.099,-72.054,172.616,27.226,154.971
C09776=1066.825,88.348,-72.072,172.617,27.229,154.971
C09777=1066.830,88.597,-72.090,172.619,27.232,154.971
C09778=1066.837,88.846,-72.108,172.620,27.234,154.972
C09779=1066.843,89.096,-72.126,172.622,27.237,154.972
C09780=1066.849,89.344,-72.145,172.623,27.240,154.973
C09781=1066.854,89.594,-72.163,172.625,27.242,154.973
C09782=1066.861,89.844,-72.182,172.626,27.245,154.973
C09783=1066.866,90.093,-72.199,172.628,27.248,154.974
C09784=1066.873,90.342,-72.218,172.629,27.251,154.974
C09785=1066.879,90.591,-72.236,172.631,27.253,154.974
C09786=1066.884,90.840,-72.255,172.632,27.256,154.975
C09787=1066.890,91.090,-72.273,172.634,27.259,154.975
C09788=1066.896,91.339,-72.291,172.635,27.261,154.976
C09789=1066.901,91.588,-72.310,172.637,27.264,154.976
C09790=1066.907,91.838,-72.328,172.638,27.267,154.976
C09791=1066.913,92.086,-72.347,172.640,27.270,154.977
C09792=1066.919,92.336,-72.365,172.641,27.273,154.977
C09793=1066.925,92.585,-72.384,172.643,27.275,154.978
C09794=1066.930,92.834,-72.402,172.644,27.278,154.978
C09795=1066.936,93.084,-72.421,172.646,27.280,154.978
C09796=1066.942,93.333,-72.440,172.647,27.283,154.979
C09797=1066.948,93.582,-72.457,172.649,27.286,154.979
C09798=1066.954,93.831,-72.476,172.650,27.289,154.979
C09799=1066.960,94.081,-72.495,172.652,27.292,154.980
C09800=1066.966,94.364,-72.516,172.653,27.295,154.980
C09801=1066.973,94.648,-72.537,172.655,27.298,154.981
C09802=1066.980,94.930,-72.558,172.657,27.301,154.981
C09803=1066.986,95.214,-72.579,172.658,27.304,154.982
C09804=1066.992,95.463,-72.598,172.660,27.307,154.982
C09805=1066.998,95.713,-72.616,172.661,27.309,154.982
C09806=1067.003,95.962,-72.635,172.663,27.312,154.983
C09807=1067.009,96.211,-72.654,172.664,27.315,154.983
C09808=1067.015,96.460,-72.672,172.666,27.318,154.984
C09809=1067.021,96.710,-72.691,172.667,27.321,154.984
C09810=1067.027,96.958,-72.709,172.669,27.323,154.984
C09811=1067.033,97.208,-72.728,172.670,27.326,154.985
C09812=1067.039,97.458,-72.746,172.672,27.328,154.985
C09813=1067.044,97.707,-72.765,172.673,27.331,154.985
C09814=1067.050,97.955,-72.784,172.675,27.334,154.986
C09815=1067.056,98.205,-72.803,172.676,27.337,154.986
C09816=1067.062,98.454,-72.822,172.678,27.340,154.987
C09817=1067.068,98.704,-72.840,172.679,27.342,154.987
C09818=1067.074,98.952,-72.858,172.681,27.345,154.987
C09819=1067.079,99.202,-72.878,172.682,27.348,154.988
C09820=1067.086,99.451,-72.896,172.684,27.350,154.988
C09821=1067.092,99.700,-72.915,172.686,27.353,154.988
C09822=1067.098,99.950,-72.934,172.688,27.356,154.989
C09823=1067.103,100.199,-72.952,172.689,27.358,154.989
C09824=1067.109,100.448,-72.971,172.691,27.361,154.990
C09825=1067.116,100.697,-72.990,172.692,27.364,154.990
C09826=1067.121,100.947,-73.009,172.694,27.367,154.990
C09827=1067.128,101.196,-73.028,172.695,27.370,154.991
C09828=1067.133,101.444,-73.046,172.697,27.372,154.991
C09829=1067.138,101.694,-73.066,172.698,27.375,154.992
C09830=1067.144,101.943,-73.085,172.700,27.377,154.992
C09831=1067.151,102.192,-73.104,172.701,27.380,154.992
C09832=1067.156,102.441,-73.123,172.703,27.383,154.993
C09833=1067.161,102.691,-73.142,172.704,27.386,154.993
C09834=1067.167,102.940,-73.160,172.706,27.389,154.993
C09835=1067.173,103.190,-73.179,172.707,27.391,154.994
C09836=1067.179,103.439,-73.198,172.709,27.394,154.994
C09837=1067.185,103.688,-73.216,172.710,27.397,154.995
C09838=1067.190,103.937,-73.236,172.712,27.400,154.995
C09839=1067.196,104.186,-73.255,172.713,27.403,154.995
C09840=1067.202,104.436,-73.274,172.715,27.405,154.996
C09841=1067.208,104.685,-73.293,172.716,27.408,154.996
C09842=1067.214,104.934,-73.312,172.718,27.411,154.997
C09843=1067.219,105.183,-73.331,172.719,27.413,154.997
C09844=1067.226,105.432,-73.350,172.721,27.416,154.997
C09845=1067.231,105.681,-73.370,172.722,27.419,154.998
C09846=1067.237,105.931,-73.389,172.724,27.422,154.998
C09847=1067.243,106.180,-73.408,172.725,27.424,154.999
C09848=1067.249,106.429,-73.427,172.727,27.427,154.999
C09849=1067.254,106.678,-73.446,172.729,27.430,154.999
C09850=1067.260,106.927,-73.465,172.730,27.432,155.000
C09851=1067.266,107.177,-73.484,172.732,27.435,155.000
C09852=1067.272,107.426,-73.503,172.734,27.438,155.000
C09853=1067.278,107.675,-73.522,172.735,27.441,155.001
C09854=1067.283,107.925,-73.541,172.737,27.444,155.001
C09855=1067.290,108.173,-73.561,172.738,27.447,155.002
C09856=1067.296,108.423,-73.580,172.740,27.449,155.002
C09857=1067.301,108.672,-73.599,172.742,27.452,155.002
C09858=1067.307,108.921,-73.618,172.743,27.454,155.003
C09859=1067.312,109.170,-73.637,172.745,27.457,155.003
C09860=1067.319,109.419,-73.656,172.746,27.460,155.004
C09861=1067.325,109.668,-73.676,172.748,27.463,155.004
C09862=1067.330,109.918,-73.695,172.749,27.465,155.004
C09863=1067.336,110.167,-73.714,172.751,27.468,155.005
C09864=1067.343,110.450,-73.736,172.752,27.471,155.005
C09865=1067.349,110.733,-73.758,172.755,27.474,155.006
C09866=1067.357,111.017,-73.780,172.756,27.477,155.006
C09867=1067.363,111.300,-73.802,172.757,27.480,155.006
C09868=1067.369,111.550,-73.821,172.760,27.483,155.007
C09869=1067.374,111.799,-73.840,172.761,27.486,155.007
C09870=1067.381,112.048,-73.859,172.763,27.488,155.008
C09871=1067.387,112.297,-73.879,172.764,27.491,155.008
C09872=1067.393,112.546,-73.898,172.766,27.494,155.008
C09873=1067.398,112.796,-73.918,172.767,27.497,155.009
C09874=1067.404,113.045,-73.938,172.769,27.500,155.009
C09875=1067.409,113.293,-73.956,172.770,27.502,155.010
C09876=1067.415,113.543,-73.976,172.772,27.505,155.010
C09877=1067.421,113.792,-73.995,172.774,27.507,155.010
C09878=1067.427,114.041,-74.015,172.775,27.510,155.011
C09879=1067.432,114.291,-74.034,172.777,27.513,155.011
C09880=1067.438,114.539,-74.054,172.778,27.516,155.011
C09881=1067.444,114.789,-74.073,172.780,27.519,155.012
C09882=1067.450,115.038,-74.093,172.781,27.521,155.012
C09883=1067.456,115.287,-74.113,172.784,27.524,155.013
C09884=1067.461,115.536,-74.132,172.785,27.527,155.013
C09885=1067.467,115.785,-74.152,172.787,27.530,155.013
C09886=1067.472,116.035,-74.172,172.788,27.533,155.014
C09887=1067.478,116.284,-74.191,172.790,27.536,155.014
C09888=1067.484,116.533,-74.211,172.791,27.538,155.015
C09889=1067.490,116.783,-74.230,172.793,27.541,155.015
C09890=1067.496,117.032,-74.250,172.794,27.544,155.015
C09891=1067.501,117.281,-74.269,172.796,27.546,155.016
C09892=1067.507,117.529,-74.289,172.797,27.549,155.016
C09893=1067.512,117.779,-74.309,172.799,27.552,155.017
C09894=1067.518,118.028,-74.329,172.800,27.554,155.017
C09895=1067.523,118.277,-74.348,172.802,27.557,155.017
C09896=1067.529,118.526,-74.368,172.804,27.560,155.018
C09897=1067.535,118.775,-74.387,172.806,27.563,155.018
C09898=1067.541,119.024,-74.407,172.807,27.566,155.019
C09899=1067.546,119.274,-74.427,172.809,27.569,155.019
C09900=1067.552,119.523,-74.447,172.810,27.571,155.019
C09901=1067.558,119.772,-74.466,172.812,27.574,155.020
C09902=1067.564,120.021,-74.486,172.813,27.577,155.020
C09903=1067.570,120.270,-74.506,172.815,27.580,155.021
C09904=1067.575,120.519,-74.525,172.816,27.582,155.021
C09905=1067.581,120.769,-74.546,172.818,27.585,155.021
C09906=1067.587,121.018,-74.565,172.819,27.588,155.022
C09907=1067.593,121.267,-74.585,172.822,27.591,155.022
C09908=1067.599,121.517,-74.605,172.823,27.593,155.022
C09909=1067.605,121.766,-74.625,172.825,27.596,155.023
C09910=1067.610,122.015,-74.645,172.826,27.599,155.023
C09911=1067.616,122.264,-74.664,172.828,27.602,155.024
C09912=1067.622,122.513,-74.684,172.829,27.605,155.024
C09913=1067.628,122.762,-74.704,172.831,27.607,155.024
C09914=1067.633,123.011,-74.723,172.833,27.610,155.025
C09915=1067.639,123.260,-74.744,172.834,27.612,155.025
C09916=1067.645,123.509,-74.764,172.837,27.615,155.025
C09917=1067.650,123.758,-74.783,172.838,27.618,155.026
C09918=1067.656,124.007,-74.803,172.840,27.621,155.026
C09919=1067.663,124.257,-74.824,172.841,27.624,155.027
C09920=1067.668,124.506,-74.844,172.843,27.627,155.027
C09921=1067.674,124.755,-74.863,172.844,27.629,155.027
C09922=1067.680,125.004,-74.883,172.846,27.632,155.028
C09923=1067.686,125.253,-74.903,172.847,27.634,155.028
C09924=1067.691,125.503,-74.923,172.849,27.637,155.029
C09925=1067.697,125.752,-74.943,172.851,27.640,155.029
C09926=1067.703,126.000,-74.963,172.853,27.643,155.029
C09927=1067.709,126.250,-74.983,172.854,27.646,155.030
C09928=1067.716,126.534,-75.006,172.856,27.648,155.030
C09929=1067.721,126.816,-75.029,172.858,27.651,155.031
C09930=1067.728,127.100,-75.051,172.860,27.655,155.031
C09931=1067.735,127.383,-75.074,172.862,27.658,155.031
C09932=1067.741,127.632,-75.095,172.864,27.661,155.032
C09933=1067.747,127.881,-75.115,172.865,27.663,155.032
C09934=1067.753,128.130,-75.135,172.867,27.666,155.033
C09935=1067.758,128.380,-75.154,172.868,27.668,155.033
C09936=1067.764,128.629,-75.174,172.870,27.671,155.033
C09937=1067.771,128.878,-75.195,172.871,27.674,155.034
C09938=1067.776,129.127,-75.215,172.873,27.677,155.034
C09939=1067.782,129.376,-75.235,172.875,27.679,155.034
C09940=1067.788,129.625,-75.255,172.877,27.682,155.035
C09941=1067.794,129.874,-75.275,172.878,27.685,155.035
C09942=1067.800,130.123,-75.296,172.880,27.688,155.036
C09943=1067.806,130.372,-75.316,172.882,27.690,155.036
C09944=1067.812,130.621,-75.336,172.883,27.693,155.036
C09945=1067.817,130.871,-75.356,172.885,27.695,155.037
C09946=1067.824,131.120,-75.376,172.887,27.698,155.037
C09947=1067.830,131.369,-75.396,172.889,27.701,155.038
C09948=1067.835,131.618,-75.417,172.890,27.704,155.038
C09949=1067.841,131.867,-75.437,172.892,27.706,155.038
C09950=1067.847,132.117,-75.457,172.893,27.709,155.039
C09951=1067.853,132.366,-75.477,172.895,27.712,155.039
C09952=1067.859,132.615,-75.497,172.897,27.715,155.039
C09953=1067.864,132.864,-75.518,172.899,27.717,155.040
C09954=1067.870,133.112,-75.538,172.900,27.720,155.040
C09955=1067.876,133.362,-75.559,172.902,27.723,155.041
C09956=1067.881,133.611,-75.579,172.903,27.726,155.041
C09957=1067.887,133.860,-75.600,172.905,27.729,155.041
C09958=1067.893,134.109,-75.621,172.907,27.732,155.042
C09959=1067.899,134.358,-75.641,172.909,27.734,155.042
C09960=1067.904,134.607,-75.661,172.911,27.737,155.042
C09961=1067.910,134.856,-75.681,172.912,27.739,155.043
C09962=1067.916,135.105,-75.702,172.914,27.742,155.043
C09963=1067.922,135.355,-75.722,172.915,27.745,155.044
C09964=1067.927,135.604,-75.743,172.917,27.748,155.044
C09965=1067.933,135.853,-75.763,172.919,27.751,155.044
C09966=1067.939,136.101,-75.784,172.921,27.753,155.045
C09967=1067.945,136.351,-75.805,172.922,27.756,155.045
C09968=1067.951,136.600,-75.825,172.924,27.758,155.046
C09969=1067.956,136.849,-75.846,172.925,27.761,155.046
C09970=1067.962,137.098,-75.865,172.928,27.764,155.046
C09971=1067.968,137.348,-75.886,172.929,27.767,155.047
C09972=1067.974,137.596,-75.908,172.931,27.770,155.047
C09973=1067.980,137.845,-75.928,172.932,27.773,155.048
C09974=1067.985,138.095,-75.949,172.934,27.775,155.048
C09975=1067.991,138.344,-75.969,172.935,27.778,155.048
C09976=1067.997,138.593,-75.989,172.938,27.781,155.049
C09977=1068.003,138.842,-76.011,172.940,27.783,155.049
C09978=1068.008,139.091,-76.031,172.941,27.786,155.049
C09979=1068.014,139.340,-76.051,172.943,27.789,155.050
C09980=1068.020,139.589,-76.073,172.944,27.792,155.050
C09981=1068.026,139.838,-76.093,172.947,27.795,155.051
C09982=1068.031,140.087,-76.113,172.948,27.797,155.051
C09983=1068.037,140.337,-76.134,172.950,27.800,155.051
C09984=1068.043,140.585,-76.156,172.951,27.803,155.052
C09985=1068.049,140.834,-76.176,172.953,27.805,155.052
C09986=1068.054,141.083,-76.196,172.955,27.808,155.053
C09987=1068.060,141.332,-76.218,172.957,27.811,155.053
C09988=1068.066,141.582,-76.238,172.958,27.814,155.053
C09989=1068.071,141.831,-76.259,172.960,27.816,155.054
C09990=1068.078,142.080,-76.280,172.961,27.819,155.054
C09991=1068.083,142.329,-76.300,172.964,27.822,155.055
C09992=1068.089,142.611,-76.325,172.965,27.825,155.055
C09993=1068.096,142.895,-76.348,172.968,27.829,155.055
C09994=1068.103,143.179,-76.372,172.969,27.831,155.056
C09995=1068.109,143.462,-76.395,172.972,27.835,155.056
C09996=1068.115,143.710,-76.417,172.973,27.838,155.057
//INST
///DATE 2021/06/17 10:55
///ATTR SC,RW,RJ
////FRAME ROBOT
///GROUP1 RB1
NOP
MOVL C00000 V=800.0 PL=0
MOVL C00001 V=800.0 PL=0
MOVL C00002 V=800.0 PL=0
MOVL C00003 V=800.0 PL=0
MOVL C00004 V=800.0 PL=0
MOVL C00005 V=800.0 PL=0
MOVL C00006 V=800.0 PL=0
MOVL C00007 V=800.0 PL=0
MOVL C00008 V=800.0 PL=0
MOVL C00009 V=800.0 PL=0
MOVL C00010 V=800.0 PL=0
MOVL C00011 V=800.0 PL=0
MOVL C00012 V=800.0 PL=0
MOVL C00013 V=800.0 PL=0
MOVL C00014 V=800.0 PL=0
MOVL C00015 V=800.0 PL=0
MOVL C00016 V=800.0 PL=0
MOVL C00017 V=800.0 PL=0
MOVL C00018 V=800.0 PL=0
MOVL C00019 V=800.0 PL=0
MOVL C00020 V=800.0 PL=0
MOVL C00021 V=800.0 PL=0
MOVL C00022 V=800.0 PL=0
MOVL C00023 V=800.0 PL=0
MOVL C00024 V=800.0 PL=0
MOVL C00025 V=800.0 PL=0
MOVL C00026 V=800.0 PL=0
MOVL C00027 V=800.0 PL=0
MOVL C00028 V=800.0 PL=0
MOVL C00029 V=800.0 PL=0
MOVL C00030 V=800.0 PL=0
MOVL C00031 V=800.0 PL=0
MOVL C00032 V=800.0 PL=0
MOVL C00033 V=800.0 PL=0
MOVL C00034 V=800.0 PL=0
MOVL C00035 V=800.0 PL=0
MOVL C00036 V=800.0 PL=0
MOVL C00037 V=800.0 PL=0
MOVL C00038 V=800.0 PL=0
MOVL C00039 V=800.0 PL=0
MOVL C00040 V=800.0 PL=0
MOVL C00041 V=800.0 PL=0
MOVL C00042 V=800.0 PL=0
MOVL C00043 V=800.0 PL=0
MOVL C00044 V=800.0 PL=0
MOVL C00045 V=800.0 PL=0
MOVL C00046 V=800.0 PL=0
MOVL C00047 V=800.0 PL=0
MOVL C00048 V=800.0 PL=0
MOVL C00049 V=800.0 PL=0
MOVL C00050 V=800.0 PL=0
MOVL C00051 V=800.0 PL=0
MOVL C00052 V=800.0 PL=0
MOVL C00053 V=800.0 PL=0
MOVL C00054 V=800.0 PL=0
MOVL C00055 V=800.0 PL=0
MOVL C00056 V=800.0 PL=0
MOVL C00057 V=800.0 PL=0
MOVL C00058 V=800.0 PL=0
MOVL C00059 V=800.0 PL=0
MOVL C00060 V=800.0 PL=0
MOVL C00061 V=800.0 PL=0
MOVL C00062 V=800.0 PL=0
MOVL C00063 V=800.0 PL=0
MOVL C00064 V=800.0 PL=0
MOVL C00065 V=800.0 PL=0
MOVL C00066 V=800.0 PL=0
MOVL C00067 V=800.0 PL=0
MOVL C00068 V=800.0 PL=0
MOVL C00069 V=800.0 PL=0
MOVL C00070 V=800.0 PL=0
MOVL C00071 V=800.0 PL=0
MOVL C00072 V=800.0 PL=0
MOVL C00073 V=800.0 PL=0
MOVL C00074 V=800.0 PL=0
MOVL C00075 V=800.0 PL=0
MOVL C00076 V=800.0 PL=0
MOVL C00077 V=800.0 PL=0
MOVL C00078 V=800.0 PL=0
MOVL C00079 V=800.0 PL=0
MOVL C00080 V=800.0 PL=0
MOVL C00081 V=800.0 PL=0
MOVL C00082 V=800.0 PL=0
MOVL C00083 V=800.0 PL=0
MOVL C00084 V=800.0 PL=0
MOVL C00085 V=800.0 PL=0
MOVL C00086 V=800.0 PL=0
MOVL C00087 V=800.0 PL=0
MOVL C00088 V=800.0 PL=0
MOVL C00089 V=800.0 PL=0
MOVL C00090 V=800.0 PL=0
MOVL C00091 V=800.0 PL=0
MOVL C00092 V=800.0 PL=0
MOVL C00093 V=800.0 PL=0
MOVL C00094 V=800.0 PL=0
MOVL C00095 V=800.0 PL=0
MOVL C00096 V=800.0 PL=0
MOVL C00097 V=800.0 PL=0
MOVL C00098 V=800.0 PL=0
MOVL C00099 V=800.0 PL=0
MOVL C00100 V=800.0 PL=0
MOVL C00101 V=800.0 PL=0
MOVL C00102 V=800.0 PL=0
MOVL C00103 V=800.0 PL=0
MOVL C00104 V=800.0 PL=0
MOVL C00105 V=800.0 PL=0
MOVL C00106 V=800.0 PL=0
MOVL C00107 V=800.0 PL=0
MOVL C00108 V=800.0 PL=0
MOVL C00109 V=800.0 PL=0
MOVL C00110 V=800.0 PL=0
MOVL C00111 V=800.0 PL=0
MOVL C00112 V=800.0 PL=0
MOVL C00113 V=800.0 PL=0
MOVL C00114 V=800.0 PL=0
MOVL C00115 V=800.0 PL=0
MOVL C00116 V=800.0 PL=0
MOVL C00117 V=800.0 PL=0
MOVL C00118 V=800.0 PL=0
MOVL C00119 V=800.0 PL=0
MOVL C00120 V=800.0 PL=0
MOVL C00121 V=800.0 PL=0
MOVL C00122 V=800.0 PL=0
MOVL C00123 V=800.0 PL=0
MOVL C00124 V=800.0 PL=0
MOVL C00125 V=800.0 PL=0
MOVL C00126 V=800.0 PL=0
MOVL C00127 V=800.0 PL=0
MOVL C00128 V=800.0 PL=0
MOVL C00129 V=800.0 PL=0
MOVL C00130 V=800.0 PL=0
MOVL C00131 V=800.0 PL=0
MOVL C00132 V=800.0 PL=0
MOVL C00133 V=800.0 PL=0
MOVL C00134 V=800.0 PL=0
MOVL C00135 V=800.0 PL=0
MOVL C00136 V=800.0 PL=0
MOVL C00137 V=800.0 PL=0
MOVL C00138 V=800.0 PL=0
MOVL C00139 V=800.0 PL=0
MOVL C00140 V=800.0 PL=0
MOVL C00141 V=800.0 PL=0
MOVL C00142 V=800.0 PL=0
MOVL C00143 V=800.0 PL=0
MOVL C00144 V=800.0 PL=0
MOVL C00145 V=800.0 PL=0
MOVL C00146 V=800.0 PL=0
MOVL C00147 V=800.0 PL=0
MOVL C00148 V=800.0 PL=0
MOVL C00149 V=800.0 PL=0
MOVL C00150 V=800.0 PL=0
MOVL C00151 V=800.0 PL=0
MOVL C00152 V=800.0 PL=0
MOVL C00153 V=800.0 PL=0
MOVL C00154 V=800.0 PL=0
MOVL C00155 V=800.0 PL=0
MOVL C00156 V=800.0 PL=0
MOVL C00157 V=800.0 PL=0
MOVL C00158 V=800.0 PL=0
MOVL C00159 V=800.0 PL=0
MOVL C00160 V=800.0 PL=0
MOVL C00161 V=800.0 PL=0
MOVL C00162 V=800.0 PL=0
MOVL C00163 V=800.0 PL=0
MOVL C00164 V=800.0 PL=0
MOVL C00165 V=800.0 PL=0
MOVL C00166 V=800.0 PL=0
MOVL C00167 V=800.0 PL=0
MOVL C00168 V=800.0 PL=0
MOVL C00169 V=800.0 PL=0
MOVL C00170 V=800.0 PL=0
MOVL C00171 V=800.0 PL=0
MOVL C00172 V=800.0 PL=0
MOVL C00173 V=800.0 PL=0
MOVL C00174 V=800.0 PL=0
MOVL C00175 V=800.0 PL=0
MOVL C00176 V=800.0 PL=0
MOVL C00177 V=800.0 PL=0
MOVL C00178 V=800.0 PL=0
MOVL C00179 V=800.0 PL=0
MOVL C00180 V=800.0 PL=0
MOVL C00181 V=800.0 PL=0
MOVL C00182 V=800.0 PL=0
MOVL C00183 V=800.0 PL=0
MOVL C00184 V=800.0 PL=0
MOVL C00185 V=800.0 PL=0
MOVL C00186 V=800.0 PL=0
MOVL C00187 V=800.0 PL=0
MOVL C00188 V=800.0 PL=0
MOVL C00189 V=800.0 PL=0
MOVL C00190 V=800.0 PL=0
MOVL C00191 V=800.0 PL=0
MOVL C00192 V=800.0 PL=0
MOVL C00193 V=800.0 PL=0
MOVL C00194 V=800.0 PL=0
MOVL C00195 V=800.0 PL=0
MOVL C00196 V=800.0 PL=0
MOVL C00197 V=800.0 PL=0
MOVL C00198 V=800.0 PL=0
MOVL C00199 V=800.0 PL=0
MOVL C00200 V=800.0 PL=0
MOVL C00201 V=800.0 PL=0
MOVL C00202 V=800.0 PL=0
MOVL C00203 V=800.0 PL=0
MOVL C00204 V=800.0 PL=0
MOVL C00205 V=800.0 PL=0
MOVL C00206 V=800.0 PL=0
MOVL C00207 V=800.0 PL=0
MOVL C00208 V=800.0 PL=0
MOVL C00209 V=800.0 PL=0
MOVL C00210 V=800.0 PL=0
MOVL C00211 V=800.0 PL=0
MOVL C00212 V=800.0 PL=0
MOVL C00213 V=800.0 PL=0
MOVL C00214 V=800.0 PL=0
MOVL C00215 V=800.0 PL=0
MOVL C00216 V=800.0 PL=0
MOVL C00217 V=800.0 PL=0
MOVL C00218 V=800.0 PL=0
MOVL C00219 V=800.0 PL=0
MOVL C00220 V=800.0 PL=0
MOVL C00221 V=800.0 PL=0
MOVL C00222 V=800.0 PL=0
MOVL C00223 V=800.0 PL=0
MOVL C00224 V=800.0 PL=0
MOVL C00225 V=800.0 PL=0
MOVL C00226 V=800.0 PL=0
MOVL C00227 V=800.0 PL=0
MOVL C00228 V=800.0 PL=0
MOVL C00229 V=800.0 PL=0
MOVL C00230 V=800.0 PL=0
MOVL C00231 V=800.0 PL=0
MOVL C00232 V=800.0 PL=0
MOVL C00233 V=800.0 PL=0
MOVL C00234 V=800.0 PL=0
MOVL C00235 V=800.0 PL=0
MOVL C00236 V=800.0 PL=0
MOVL C00237 V=800.0 PL=0
MOVL C00238 V=800.0 PL=0
MOVL C00239 V=800.0 PL=0
MOVL C00240 V=800.0 PL=0
MOVL C00241 V=800.0 PL=0
MOVL C00242 V=800.0 PL=0
MOVL C00243 V=800.0 PL=0
MOVL C00244 V=800.0 PL=0
MOVL C00245 V=800.0 PL=0
MOVL C00246 V=800.0 PL=0
MOVL C00247 V=800.0 PL=0
MOVL C00248 V=800.0 PL=0
MOVL C00249 V=800.0 PL=0
MOVL C00250 V=800.0 PL=0
MOVL C00251 V=800.0 PL=0
MOVL C00252 V=800.0 PL=0
MOVL C00253 V=800.0 PL=0
MOVL C00254 V=800.0 PL=0
MOVL C00255 V=800.0 PL=0
MOVL C00256 V=800.0 PL=0
MOVL C00257 V=800.0 PL=0
MOVL C00258 V=800.0 PL=0
MOVL C00259 V=800.0 PL=0
MOVL C00260 V=800.0 PL=0
MOVL C00261 V=800.0 PL=0
MOVL C00262 V=800.0 PL=0
MOVL C00263 V=800.0 PL=0
MOVL C00264 V=800.0 PL=0
MOVL C00265 V=800.0 PL=0
MOVL C00266 V=800.0 PL=0
MOVL C00267 V=800.0 PL=0
MOVL C00268 V=800.0 PL=0
MOVL C00269 V=800.0 PL=0
MOVL C00270 V=800.0 PL=0
MOVL C00271 V=800.0 PL=0
MOVL C00272 V=800.0 PL=0
MOVL C00273 V=800.0 PL=0
MOVL C00274 V=800.0 PL=0
MOVL C00275 V=800.0 PL=0
MOVL C00276 V=800.0 PL=0
MOVL C00277 V=800.0 PL=0
MOVL C00278 V=800.0 PL=0
MOVL C00279 V=800.0 PL=0
MOVL C00280 V=800.0 PL=0
MOVL C00281 V=800.0 PL=0
MOVL C00282 V=800.0 PL=0
MOVL C00283 V=800.0 PL=0
MOVL C00284 V=800.0 PL=0
MOVL C00285 V=800.0 PL=0
MOVL C00286 V=800.0 PL=0
MOVL C00287 V=800.0 PL=0
MOVL C00288 V=800.0 PL=0
MOVL C00289 V=800.0 PL=0
MOVL C00290 V=800.0 PL=0
MOVL C00291 V=800.0 PL=0
MOVL C00292 V=800.0 PL=0
MOVL C00293 V=800.0 PL=0
MOVL C00294 V=800.0 PL=0
MOVL C00295 V=800.0 PL=0
MOVL C00296 V=800.0 PL=0
MOVL C00297 V=800.0 PL=0
MOVL C00298 V=800.0 PL=0
MOVL C00299 V=800.0 PL=0
MOVL C00300 V=800.0 PL=0
MOVL C00301 V=800.0 PL=0
MOVL C00302 V=800.0 PL=0
MOVL C00303 V=800.0 PL=0
MOVL C00304 V=800.0 PL=0
MOVL C00305 V=800.0 PL=0
MOVL C00306 V=800.0 PL=0
MOVL C00307 V=800.0 PL=0
MOVL C00308 V=800.0 PL=0
MOVL C00309 V=800.0 PL=0
MOVL C00310 V=800.0 PL=0
MOVL C00311 V=800.0 PL=0
MOVL C00312 V=800.0 PL=0
MOVL C00313 V=800.0 PL=0
MOVL C00314 V=800.0 PL=0
MOVL C00315 V=800.0 PL=0
MOVL C00316 V=800.0 PL=0
MOVL C00317 V=800.0 PL=0
MOVL C00318 V=800.0 PL=0
MOVL C00319 V=800.0 PL=0
MOVL C00320 V=800.0 PL=0
MOVL C00321 V=800.0 PL=0
MOVL C00322 V=800.0 PL=0
MOVL C00323 V=800.0 PL=0
MOVL C00324 V=800.0 PL=0
MOVL C00325 V=800.0 PL=0
MOVL C00326 V=800.0 PL=0
MOVL C00327 V=800.0 PL=0
MOVL C00328 V=800.0 PL=0
MOVL C00329 V=800.0 PL=0
MOVL C00330 V=800.0 PL=0
MOVL C00331 V=800.0 PL=0
MOVL C00332 V=800.0 PL=0
MOVL C00333 V=800.0 PL=0
MOVL C00334 V=800.0 PL=0
MOVL C00335 V=800.0 PL=0
MOVL C00336 V=800.0 PL=0
MOVL C00337 V=800.0 PL=0
MOVL C00338 V=800.0 PL=0
MOVL C00339 V=800.0 PL=0
MOVL C00340 V=800.0 PL=0
MOVL C00341 V=800.0 PL=0
MOVL C00342 V=800.0 PL=0
MOVL C00343 V=800.0 PL=0
MOVL C00344 V=800.0 PL=0
MOVL C00345 V=800.0 PL=0
MOVL C00346 V=800.0 PL=0
MOVL C00347 V=800.0 PL=0
MOVL C00348 V=800.0 PL=0
MOVL C00349 V=800.0 PL=0
MOVL C00350 V=800.0 PL=0
MOVL C00351 V=800.0 PL=0
MOVL C00352 V=800.0 PL=0
MOVL C00353 V=800.0 PL=0
MOVL C00354 V=800.0 PL=0
MOVL C00355 V=800.0 PL=0
MOVL C00356 V=800.0 PL=0
MOVL C00357 V=800.0 PL=0
MOVL C00358 V=800.0 PL=0
MOVL C00359 V=800.0 PL=0
MOVL C00360 V=800.0 PL=0
MOVL C00361 V=800.0 PL=0
MOVL C00362 V=800.0 PL=0
MOVL C00363 V=800.0 PL=0
MOVL C00364 V=800.0 PL=0
MOVL C00365 V=800.0 PL=0
MOVL C00366 V=800.0 PL=0
MOVL C00367 V=800.0 PL=0
MOVL C00368 V=800.0 PL=0
MOVL C00369 V=800.0 PL=0
MOVL C00370 V=800.0 PL=0
MOVL C00371 V=800.0 PL=0
MOVL C00372 V=800.0 PL=0
MOVL C00373 V=800.0 PL=0
MOVL C00374 V=800.0 PL=0
MOVL C00375 V=800.0 PL=0
MOVL C00376 V=800.0 PL=0
MOVL C00377 V=800.0 PL=0
MOVL C00378 V=800.0 PL=0
MOVL C00379 V=800.0 PL=0
MOVL C00380 V=800.0 PL=0
MOVL C00381 V=800.0 PL=0
MOVL C00382 V=800.0 PL=0
MOVL C00383 V=800.0 PL=0
MOVL C00384 V=800.0 PL=0
MOVL C00385 V=800.0 PL=0
MOVL C00386 V=800.0 PL=0
MOVL C00387 V=800.0 PL=0
MOVL C00388 V=800.0 PL=0
MOVL C00389 V=800.0 PL=0
MOVL C00390 V=800.0 PL=0
MOVL C00391 V=800.0 PL=0
MOVL C00392 V=800.0 PL=0
MOVL C00393 V=800.0 PL=0
MOVL C00394 V=800.0 PL=0
MOVL C00395 V=800.0 PL=0
MOVL C00396 V=800.0 PL=0
MOVL C00397 V=800.0 PL=0
MOVL C00398 V=800.0 PL=0
MOVL C00399 V=800.0 PL=0
MOVL C00400 V=800.0 PL=0
MOVL C00401 V=800.0 PL=0
MOVL C00402 V=800.0 PL=0
MOVL C00403 V=800.0 PL=0
MOVL C00404 V=800.0 PL=0
MOVL C00405 V=800.0 PL=0
MOVL C00406 V=800.0 PL=0
MOVL C00407 V=800.0 PL=0
MOVL C00408 V=800.0 PL=0
MOVL C00409 V=800.0 PL=0
MOVL C00410 V=800.0 PL=0
MOVL C00411 V=800.0 PL=0
MOVL C00412 V=800.0 PL=0
MOVL C00413 V=800.0 PL=0
MOVL C00414 V=800.0 PL=0
MOVL C00415 V=800.0 PL=0
MOVL C00416 V=800.0 PL=0
MOVL C00417 V=800.0 PL=0
MOVL C00418 V=800.0 PL=0
MOVL C00419 V=800.0 PL=0
MOVL C00420 V=800.0 PL=0
MOVL C00421 V=800.0 PL=0
MOVL C00422 V=800.0 PL=0
MOVL C00423 V=800.0 PL=0
MOVL C00424 V=800.0 PL=0
MOVL C00425 V=800.0 PL=0
MOVL C00426 V=800.0 PL=0
MOVL C00427 V=800.0 PL=0
MOVL C00428 V=800.0 PL=0
MOVL C00429 V=800.0 PL=0
MOVL C00430 V=800.0 PL=0
MOVL C00431 V=800.0 PL=0
MOVL C00432 V=800.0 PL=0
MOVL C00433 V=800.0 PL=0
MOVL C00434 V=800.0 PL=0
MOVL C00435 V=800.0 PL=0
MOVL C00436 V=800.0 PL=0
MOVL C00437 V=800.0 PL=0
MOVL C00438 V=800.0 PL=0
MOVL C00439 V=800.0 PL=0
MOVL C00440 V=800.0 PL=0
MOVL C00441 V=800.0 PL=0
MOVL C00442 V=800.0 PL=0
MOVL C00443 V=800.0 PL=0
MOVL C00444 V=800.0 PL=0
MOVL C00445 V=800.0 PL=0
MOVL C00446 V=800.0 PL=0
MOVL C00447 V=800.0 PL=0
MOVL C00448 V=800.0 PL=0
MOVL C00449 V=800.0 PL=0
MOVL C00450 V=800.0 PL=0
MOVL C00451 V=800.0 PL=0
MOVL C00452 V=800.0 PL=0
MOVL C00453 V=800.0 PL=0
MOVL C00454 V=800.0 PL=0
MOVL C00455 V=800.0 PL=0
MOVL C00456 V=800.0 PL=0
MOVL C00457 V=800.0 PL=0
MOVL C00458 V=800.0 PL=0
MOVL C00459 V=800.0 PL=0
MOVL C00460 V=800.0 PL=0
MOVL C00461 V=800.0 PL=0
MOVL C00462 V=800.0 PL=0
MOVL C00463 V=800.0 PL=0
MOVL C00464 V=800.0 PL=0
MOVL C00465 V=800.0 PL=0
MOVL C00466 V=800.0 PL=0
MOVL C00467 V=800.0 PL=0
MOVL C00468 V=800.0 PL=0
MOVL C00469 V=800.0 PL=0
MOVL C00470 V=800.0 PL=0
MOVL C00471 V=800.0 PL=0
MOVL C00472 V=800.0 PL=0
MOVL C00473 V=800.0 PL=0
MOVL C00474 V=800.0 PL=0
MOVL C00475 V=800.0 PL=0
MOVL C00476 V=800.0 PL=0
MOVL C00477 V=800.0 PL=0
MOVL C00478 V=800.0 PL=0
MOVL C00479 V=800.0 PL=0
MOVL C00480 V=800.0 PL=0
MOVL C00481 V=800.0 PL=0
MOVL C00482 V=800.0 PL=0
MOVL C00483 V=800.0 PL=0
MOVL C00484 V=800.0 PL=0
MOVL C00485 V=800.0 PL=0
MOVL C00486 V=800.0 PL=0
MOVL C00487 V=800.0 PL=0
MOVL C00488 V=800.0 PL=0
MOVL C00489 V=800.0 PL=0
MOVL C00490 V=800.0 PL=0
MOVL C00491 V=800.0 PL=0
MOVL C00492 V=800.0 PL=0
MOVL C00493 V=800.0 PL=0
MOVL C00494 V=800.0 PL=0
MOVL C00495 V=800.0 PL=0
MOVL C00496 V=800.0 PL=0
MOVL C00497 V=800.0 PL=0
MOVL C00498 V=800.0 PL=0
MOVL C00499 V=800.0 PL=0
MOVL C00500 V=800.0 PL=0
MOVL C00501 V=800.0 PL=0
MOVL C00502 V=800.0 PL=0
MOVL C00503 V=800.0 PL=0
MOVL C00504 V=800.0 PL=0
MOVL C00505 V=800.0 PL=0
MOVL C00506 V=800.0 PL=0
MOVL C00507 V=800.0 PL=0
MOVL C00508 V=800.0 PL=0
MOVL C00509 V=800.0 PL=0
MOVL C00510 V=800.0 PL=0
MOVL C00511 V=800.0 PL=0
MOVL C00512 V=800.0 PL=0
MOVL C00513 V=800.0 PL=0
MOVL C00514 V=800.0 PL=0
MOVL C00515 V=800.0 PL=0
MOVL C00516 V=800.0 PL=0
MOVL C00517 V=800.0 PL=0
MOVL C00518 V=800.0 PL=0
MOVL C00519 V=800.0 PL=0
MOVL C00520 V=800.0 PL=0
MOVL C00521 V=800.0 PL=0
MOVL C00522 V=800.0 PL=0
MOVL C00523 V=800.0 PL=0
MOVL C00524 V=800.0 PL=0
MOVL C00525 V=800.0 PL=0
MOVL C00526 V=800.0 PL=0
MOVL C00527 V=800.0 PL=0
MOVL C00528 V=800.0 PL=0
MOVL C00529 V=800.0 PL=0
MOVL C00530 V=800.0 PL=0
MOVL C00531 V=800.0 PL=0
MOVL C00532 V=800.0 PL=0
MOVL C00533 V=800.0 PL=0
MOVL C00534 V=800.0 PL=0
MOVL C00535 V=800.0 PL=0
MOVL C00536 V=800.0 PL=0
MOVL C00537 V=800.0 PL=0
MOVL C00538 V=800.0 PL=0
MOVL C00539 V=800.0 PL=0
MOVL C00540 V=800.0 PL=0
MOVL C00541 V=800.0 PL=0
MOVL C00542 V=800.0 PL=0
MOVL C00543 V=800.0 PL=0
MOVL C00544 V=800.0 PL=0
MOVL C00545 V=800.0 PL=0
MOVL C00546 V=800.0 PL=0
MOVL C00547 V=800.0 PL=0
MOVL C00548 V=800.0 PL=0
MOVL C00549 V=800.0 PL=0
MOVL C00550 V=800.0 PL=0
MOVL C00551 V=800.0 PL=0
MOVL C00552 V=800.0 PL=0
MOVL C00553 V=800.0 PL=0
MOVL C00554 V=800.0 PL=0
MOVL C00555 V=800.0 PL=0
MOVL C00556 V=800.0 PL=0
MOVL C00557 V=800.0 PL=0
MOVL C00558 V=800.0 PL=0
MOVL C00559 V=800.0 PL=0
MOVL C00560 V=800.0 PL=0
MOVL C00561 V=800.0 PL=0
MOVL C00562 V=800.0 PL=0
MOVL C00563 V=800.0 PL=0
MOVL C00564 V=800.0 PL=0
MOVL C00565 V=800.0 PL=0
MOVL C00566 V=800.0 PL=0
MOVL C00567 V=800.0 PL=0
MOVL C00568 V=800.0 PL=0
MOVL C00569 V=800.0 PL=0
MOVL C00570 V=800.0 PL=0
MOVL C00571 V=800.0 PL=0
MOVL C00572 V=800.0 PL=0
MOVL C00573 V=800.0 PL=0
MOVL C00574 V=800.0 PL=0
MOVL C00575 V=800.0 PL=0
MOVL C00576 V=800.0 PL=0
MOVL C00577 V=800.0 PL=0
MOVL C00578 V=800.0 PL=0
MOVL C00579 V=800.0 PL=0
MOVL C00580 V=800.0 PL=0
MOVL C00581 V=800.0 PL=0
MOVL C00582 V=800.0 PL=0
MOVL C00583 V=800.0 PL=0
MOVL C00584 V=800.0 PL=0
MOVL C00585 V=800.0 PL=0
MOVL C00586 V=800.0 PL=0
MOVL C00587 V=800.0 PL=0
MOVL C00588 V=800.0 PL=0
MOVL C00589 V=800.0 PL=0
MOVL C00590 V=800.0 PL=0
MOVL C00591 V=800.0 PL=0
MOVL C00592 V=800.0 PL=0
MOVL C00593 V=800.0 PL=0
MOVL C00594 V=800.0 PL=0
MOVL C00595 V=800.0 PL=0
MOVL C00596 V=800.0 PL=0
MOVL C00597 V=800.0 PL=0
MOVL C00598 V=800.0 PL=0
MOVL C00599 V=800.0 PL=0
MOVL C00600 V=800.0 PL=0
MOVL C00601 V=800.0 PL=0
MOVL C00602 V=800.0 PL=0
MOVL C00603 V=800.0 PL=0
MOVL C00604 V=800.0 PL=0
MOVL C00605 V=800.0 PL=0
MOVL C00606 V=800.0 PL=0
MOVL C00607 V=800.0 PL=0
MOVL C00608 V=800.0 PL=0
MOVL C00609 V=800.0 PL=0
MOVL C00610 V=800.0 PL=0
MOVL C00611 V=800.0 PL=0
MOVL C00612 V=800.0 PL=0
MOVL C00613 V=800.0 PL=0
MOVL C00614 V=800.0 PL=0
MOVL C00615 V=800.0 PL=0
MOVL C00616 V=800.0 PL=0
MOVL C00617 V=800.0 PL=0
MOVL C00618 V=800.0 PL=0
MOVL C00619 V=800.0 PL=0
MOVL C00620 V=800.0 PL=0
MOVL C00621 V=800.0 PL=0
MOVL C00622 V=800.0 PL=0
MOVL C00623 V=800.0 PL=0
MOVL C00624 V=800.0 PL=0
MOVL C00625 V=800.0 PL=0
MOVL C00626 V=800.0 PL=0
MOVL C00627 V=800.0 PL=0
MOVL C00628 V=800.0 PL=0
MOVL C00629 V=800.0 PL=0
MOVL C00630 V=800.0 PL=0
MOVL C00631 V=800.0 PL=0
MOVL C00632 V=800.0 PL=0
MOVL C00633 V=800.0 PL=0
MOVL C00634 V=800.0 PL=0
MOVL C00635 V=800.0 PL=0
MOVL C00636 V=800.0 PL=0
MOVL C00637 V=800.0 PL=0
MOVL C00638 V=800.0 PL=0
MOVL C00639 V=800.0 PL=0
MOVL C00640 V=800.0 PL=0
MOVL C00641 V=800.0 PL=0
MOVL C00642 V=800.0 PL=0
MOVL C00643 V=800.0 PL=0
MOVL C00644 V=800.0 PL=0
MOVL C00645 V=800.0 PL=0
MOVL C00646 V=800.0 PL=0
MOVL C00647 V=800.0 PL=0
MOVL C00648 V=800.0 PL=0
MOVL C00649 V=800.0 PL=0
MOVL C00650 V=800.0 PL=0
MOVL C00651 V=800.0 PL=0
MOVL C00652 V=800.0 PL=0
MOVL C00653 V=800.0 PL=0
MOVL C00654 V=800.0 PL=0
MOVL C00655 V=800.0 PL=0
MOVL C00656 V=800.0 PL=0
MOVL C00657 V=800.0 PL=0
MOVL C00658 V=800.0 PL=0
MOVL C00659 V=800.0 PL=0
MOVL C00660 V=800.0 PL=0
MOVL C00661 V=800.0 PL=0
MOVL C00662 V=800.0 PL=0
MOVL C00663 V=800.0 PL=0
MOVL C00664 V=800.0 PL=0
MOVL C00665 V=800.0 PL=0
MOVL C00666 V=800.0 PL=0
MOVL C00667 V=800.0 PL=0
MOVL C00668 V=800.0 PL=0
MOVL C00669 V=800.0 PL=0
MOVL C00670 V=800.0 PL=0
MOVL C00671 V=800.0 PL=0
MOVL C00672 V=800.0 PL=0
MOVL C00673 V=800.0 PL=0
MOVL C00674 V=800.0 PL=0
MOVL C00675 V=800.0 PL=0
MOVL C00676 V=800.0 PL=0
MOVL C00677 V=800.0 PL=0
MOVL C00678 V=800.0 PL=0
MOVL C00679 V=800.0 PL=0
MOVL C00680 V=800.0 PL=0
MOVL C00681 V=800.0 PL=0
MOVL C00682 V=800.0 PL=0
MOVL C00683 V=800.0 PL=0
MOVL C00684 V=800.0 PL=0
MOVL C00685 V=800.0 PL=0
MOVL C00686 V=800.0 PL=0
MOVL C00687 V=800.0 PL=0
MOVL C00688 V=800.0 PL=0
MOVL C00689 V=800.0 PL=0
MOVL C00690 V=800.0 PL=0
MOVL C00691 V=800.0 PL=0
MOVL C00692 V=800.0 PL=0
MOVL C00693 V=800.0 PL=0
MOVL C00694 V=800.0 PL=0
MOVL C00695 V=800.0 PL=0
MOVL C00696 V=800.0 PL=0
MOVL C00697 V=800.0 PL=0
MOVL C00698 V=800.0 PL=0
MOVL C00699 V=800.0 PL=0
MOVL C00700 V=800.0 PL=0
MOVL C00701 V=800.0 PL=0
MOVL C00702 V=800.0 PL=0
MOVL C00703 V=800.0 PL=0
MOVL C00704 V=800.0 PL=0
MOVL C00705 V=800.0 PL=0
MOVL C00706 V=800.0 PL=0
MOVL C00707 V=800.0 PL=0
MOVL C00708 V=800.0 PL=0
MOVL C00709 V=800.0 PL=0
MOVL C00710 V=800.0 PL=0
MOVL C00711 V=800.0 PL=0
MOVL C00712 V=800.0 PL=0
MOVL C00713 V=800.0 PL=0
MOVL C00714 V=800.0 PL=0
MOVL C00715 V=800.0 PL=0
MOVL C00716 V=800.0 PL=0
MOVL C00717 V=800.0 PL=0
MOVL C00718 V=800.0 PL=0
MOVL C00719 V=800.0 PL=0
MOVL C00720 V=800.0 PL=0
MOVL C00721 V=800.0 PL=0
MOVL C00722 V=800.0 PL=0
MOVL C00723 V=800.0 PL=0
MOVL C00724 V=800.0 PL=0
MOVL C00725 V=800.0 PL=0
MOVL C00726 V=800.0 PL=0
MOVL C00727 V=800.0 PL=0
MOVL C00728 V=800.0 PL=0
MOVL C00729 V=800.0 PL=0
MOVL C00730 V=800.0 PL=0
MOVL C00731 V=800.0 PL=0
MOVL C00732 V=800.0 PL=0
MOVL C00733 V=800.0 PL=0
MOVL C00734 V=800.0 PL=0
MOVL C00735 V=800.0 PL=0
MOVL C00736 V=800.0 PL=0
MOVL C00737 V=800.0 PL=0
MOVL C00738 V=800.0 PL=0
MOVL C00739 V=800.0 PL=0
MOVL C00740 V=800.0 PL=0
MOVL C00741 V=800.0 PL=0
MOVL C00742 V=800.0 PL=0
MOVL C00743 V=800.0 PL=0
MOVL C00744 V=800.0 PL=0
MOVL C00745 V=800.0 PL=0
MOVL C00746 V=800.0 PL=0
MOVL C00747 V=800.0 PL=0
MOVL C00748 V=800.0 PL=0
MOVL C00749 V=800.0 PL=0
MOVL C00750 V=800.0 PL=0
MOVL C00751 V=800.0 PL=0
MOVL C00752 V=800.0 PL=0
MOVL C00753 V=800.0 PL=0
MOVL C00754 V=800.0 PL=0
MOVL C00755 V=800.0 PL=0
MOVL C00756 V=800.0 PL=0
MOVL C00757 V=800.0 PL=0
MOVL C00758 V=800.0 PL=0
MOVL C00759 V=800.0 PL=0
MOVL C00760 V=800.0 PL=0
MOVL C00761 V=800.0 PL=0
MOVL C00762 V=800.0 PL=0
MOVL C00763 V=800.0 PL=0
MOVL C00764 V=800.0 PL=0
MOVL C00765 V=800.0 PL=0
MOVL C00766 V=800.0 PL=0
MOVL C00767 V=800.0 PL=0
MOVL C00768 V=800.0 PL=0
MOVL C00769 V=800.0 PL=0
MOVL C00770 V=800.0 PL=0
MOVL C00771 V=800.0 PL=0
MOVL C00772 V=800.0 PL=0
MOVL C00773 V=800.0 PL=0
MOVL C00774 V=800.0 PL=0
MOVL C00775 V=800.0 PL=0
MOVL C00776 V=800.0 PL=0
MOVL C00777 V=800.0 PL=0
MOVL C00778 V=800.0 PL=0
MOVL C00779 V=800.0 PL=0
MOVL C00780 V=800.0 PL=0
MOVL C00781 V=800.0 PL=0
MOVL C00782 V=800.0 PL=0
MOVL C00783 V=800.0 PL=0
MOVL C00784 V=800.0 PL=0
MOVL C00785 V=800.0 PL=0
MOVL C00786 V=800.0 PL=0
MOVL C00787 V=800.0 PL=0
MOVL C00788 V=800.0 PL=0
MOVL C00789 V=800.0 PL=0
MOVL C00790 V=800.0 PL=0
MOVL C00791 V=800.0 PL=0
MOVL C00792 V=800.0 PL=0
MOVL C00793 V=800.0 PL=0
MOVL C00794 V=800.0 PL=0
MOVL C00795 V=800.0 PL=0
MOVL C00796 V=800.0 PL=0
MOVL C00797 V=800.0 PL=0
MOVL C00798 V=800.0 PL=0
MOVL C00799 V=800.0 PL=0
MOVL C00800 V=800.0 PL=0
MOVL C00801 V=800.0 PL=0
MOVL C00802 V=800.0 PL=0
MOVL C00803 V=800.0 PL=0
MOVL C00804 V=800.0 PL=0
MOVL C00805 V=800.0 PL=0
MOVL C00806 V=800.0 PL=0
MOVL C00807 V=800.0 PL=0
MOVL C00808 V=800.0 PL=0
MOVL C00809 V=800.0 PL=0
MOVL C00810 V=800.0 PL=0
MOVL C00811 V=800.0 PL=0
MOVL C00812 V=800.0 PL=0
MOVL C00813 V=800.0 PL=0
MOVL C00814 V=800.0 PL=0
MOVL C00815 V=800.0 PL=0
MOVL C00816 V=800.0 PL=0
MOVL C00817 V=800.0 PL=0
MOVL C00818 V=800.0 PL=0
MOVL C00819 V=800.0 PL=0
MOVL C00820 V=800.0 PL=0
MOVL C00821 V=800.0 PL=0
MOVL C00822 V=800.0 PL=0
MOVL C00823 V=800.0 PL=0
MOVL C00824 V=800.0 PL=0
MOVL C00825 V=800.0 PL=0
MOVL C00826 V=800.0 PL=0
MOVL C00827 V=800.0 PL=0
MOVL C00828 V=800.0 PL=0
MOVL C00829 V=800.0 PL=0
MOVL C00830 V=800.0 PL=0
MOVL C00831 V=800.0 PL=0
MOVL C00832 V=800.0 PL=0
MOVL C00833 V=800.0 PL=0
MOVL C00834 V=800.0 PL=0
MOVL C00835 V=800.0 PL=0
MOVL C00836 V=800.0 PL=0
MOVL C00837 V=800.0 PL=0
MOVL C00838 V=800.0 PL=0
MOVL C00839 V=800.0 PL=0
MOVL C00840 V=800.0 PL=0
MOVL C00841 V=800.0 PL=0
MOVL C00842 V=800.0 PL=0
MOVL C00843 V=800.0 PL=0
MOVL C00844 V=800.0 PL=0
MOVL C00845 V=800.0 PL=0
MOVL C00846 V=800.0 PL=0
MOVL C00847 V=800.0 PL=0
MOVL C00848 V=800.0 PL=0
MOVL C00849 V=800.0 PL=0
MOVL C00850 V=800.0 PL=0
MOVL C00851 V=800.0 PL=0
MOVL C00852 V=800.0 PL=0
MOVL C00853 V=800.0 PL=0
MOVL C00854 V=800.0 PL=0
MOVL C00855 V=800.0 PL=0
MOVL C00856 V=800.0 PL=0
MOVL C00857 V=800.0 PL=0
MOVL C00858 V=800.0 PL=0
MOVL C00859 V=800.0 PL=0
MOVL C00860 V=800.0 PL=0
MOVL C00861 V=800.0 PL=0
MOVL C00862 V=800.0 PL=0
MOVL C00863 V=800.0 PL=0
MOVL C00864 V=800.0 PL=0
MOVL C00865 V=800.0 PL=0
MOVL C00866 V=800.0 PL=0
MOVL C00867 V=800.0 PL=0
MOVL C00868 V=800.0 PL=0
MOVL C00869 V=800.0 PL=0
MOVL C00870 V=800.0 PL=0
MOVL C00871 V=800.0 PL=0
MOVL C00872 V=800.0 PL=0
MOVL C00873 V=800.0 PL=0
MOVL C00874 V=800.0 PL=0
MOVL C00875 V=800.0 PL=0
MOVL C00876 V=800.0 PL=0
MOVL C00877 V=800.0 PL=0
MOVL C00878 V=800.0 PL=0
MOVL C00879 V=800.0 PL=0
MOVL C00880 V=800.0 PL=0
MOVL C00881 V=800.0 PL=0
MOVL C00882 V=800.0 PL=0
MOVL C00883 V=800.0 PL=0
MOVL C00884 V=800.0 PL=0
MOVL C00885 V=800.0 PL=0
MOVL C00886 V=800.0 PL=0
MOVL C00887 V=800.0 PL=0
MOVL C00888 V=800.0 PL=0
MOVL C00889 V=800.0 PL=0
MOVL C00890 V=800.0 PL=0
MOVL C00891 V=800.0 PL=0
MOVL C00892 V=800.0 PL=0
MOVL C00893 V=800.0 PL=0
MOVL C00894 V=800.0 PL=0
MOVL C00895 V=800.0 PL=0
MOVL C00896 V=800.0 PL=0
MOVL C00897 V=800.0 PL=0
MOVL C00898 V=800.0 PL=0
MOVL C00899 V=800.0 PL=0
MOVL C00900 V=800.0 PL=0
MOVL C00901 V=800.0 PL=0
MOVL C00902 V=800.0 PL=0
MOVL C00903 V=800.0 PL=0
MOVL C00904 V=800.0 PL=0
MOVL C00905 V=800.0 PL=0
MOVL C00906 V=800.0 PL=0
MOVL C00907 V=800.0 PL=0
MOVL C00908 V=800.0 PL=0
MOVL C00909 V=800.0 PL=0
MOVL C00910 V=800.0 PL=0
MOVL C00911 V=800.0 PL=0
MOVL C00912 V=800.0 PL=0
MOVL C00913 V=800.0 PL=0
MOVL C00914 V=800.0 PL=0
MOVL C00915 V=800.0 PL=0
MOVL C00916 V=800.0 PL=0
MOVL C00917 V=800.0 PL=0
MOVL C00918 V=800.0 PL=0
MOVL C00919 V=800.0 PL=0
MOVL C00920 V=800.0 PL=0
MOVL C00921 V=800.0 PL=0
MOVL C00922 V=800.0 PL=0
MOVL C00923 V=800.0 PL=0
MOVL C00924 V=800.0 PL=0
MOVL C00925 V=800.0 PL=0
MOVL C00926 V=800.0 PL=0
MOVL C00927 V=800.0 PL=0
MOVL C00928 V=800.0 PL=0
MOVL C00929 V=800.0 PL=0
MOVL C00930 V=800.0 PL=0
MOVL C00931 V=800.0 PL=0
MOVL C00932 V=800.0 PL=0
MOVL C00933 V=800.0 PL=0
MOVL C00934 V=800.0 PL=0
MOVL C00935 V=800.0 PL=0
MOVL C00936 V=800.0 PL=0
MOVL C00937 V=800.0 PL=0
MOVL C00938 V=800.0 PL=0
MOVL C00939 V=800.0 PL=0
MOVL C00940 V=800.0 PL=0
MOVL C00941 V=800.0 PL=0
MOVL C00942 V=800.0 PL=0
MOVL C00943 V=800.0 PL=0
MOVL C00944 V=800.0 PL=0
MOVL C00945 V=800.0 PL=0
MOVL C00946 V=800.0 PL=0
MOVL C00947 V=800.0 PL=0
MOVL C00948 V=800.0 PL=0
MOVL C00949 V=800.0 PL=0
MOVL C00950 V=800.0 PL=0
MOVL C00951 V=800.0 PL=0
MOVL C00952 V=800.0 PL=0
MOVL C00953 V=800.0 PL=0
MOVL C00954 V=800.0 PL=0
MOVL C00955 V=800.0 PL=0
MOVL C00956 V=800.0 PL=0
MOVL C00957 V=800.0 PL=0
MOVL C00958 V=800.0 PL=0
MOVL C00959 V=800.0 PL=0
MOVL C00960 V=800.0 PL=0
MOVL C00961 V=800.0 PL=0
MOVL C00962 V=800.0 PL=0
MOVL C00963 V=800.0 PL=0
MOVL C00964 V=800.0 PL=0
MOVL C00965 V=800.0 PL=0
MOVL C00966 V=800.0 PL=0
MOVL C00967 V=800.0 PL=0
MOVL C00968 V=800.0 PL=0
MOVL C00969 V=800.0 PL=0
MOVL C00970 V=800.0 PL=0
MOVL C00971 V=800.0 PL=0
MOVL C00972 V=800.0 PL=0
MOVL C00973 V=800.0 PL=0
MOVL C00974 V=800.0 PL=0
MOVL C00975 V=800.0 PL=0
MOVL C00976 V=800.0 PL=0
MOVL C00977 V=800.0 PL=0
MOVL C00978 V=800.0 PL=0
MOVL C00979 V=800.0 PL=0
MOVL C00980 V=800.0 PL=0
MOVL C00981 V=800.0 PL=0
MOVL C00982 V=800.0 PL=0
MOVL C00983 V=800.0 PL=0
MOVL C00984 V=800.0 PL=0
MOVL C00985 V=800.0 PL=0
MOVL C00986 V=800.0 PL=0
MOVL C00987 V=800.0 PL=0
MOVL C00988 V=800.0 PL=0
MOVL C00989 V=800.0 PL=0
MOVL C00990 V=800.0 PL=0
MOVL C00991 V=800.0 PL=0
MOVL C00992 V=800.0 PL=0
MOVL C00993 V=800.0 PL=0
MOVL C00994 V=800.0 PL=0
MOVL C00995 V=800.0 PL=0
MOVL C00996 V=800.0 PL=0
MOVL C00997 V=800.0 PL=0
MOVL C00998 V=800.0 PL=0
MOVL C00999 V=800.0 PL=0
MOVL C01000 V=800.0 PL=0
MOVL C01001 V=800.0 PL=0
MOVL C01002 V=800.0 PL=0
MOVL C01003 V=800.0 PL=0
MOVL C01004 V=800.0 PL=0
MOVL C01005 V=800.0 PL=0
MOVL C01006 V=800.0 PL=0
MOVL C01007 V=800.0 PL=0
MOVL C01008 V=800.0 PL=0
MOVL C01009 V=800.0 PL=0
MOVL C01010 V=800.0 PL=0
MOVL C01011 V=800.0 PL=0
MOVL C01012 V=800.0 PL=0
MOVL C01013 V=800.0 PL=0
MOVL C01014 V=800.0 PL=0
MOVL C01015 V=800.0 PL=0
MOVL C01016 V=800.0 PL=0
MOVL C01017 V=800.0 PL=0
MOVL C01018 V=800.0 PL=0
MOVL C01019 V=800.0 PL=0
MOVL C01020 V=800.0 PL=0
MOVL C01021 V=800.0 PL=0
MOVL C01022 V=800.0 PL=0
MOVL C01023 V=800.0 PL=0
MOVL C01024 V=800.0 PL=0
MOVL C01025 V=800.0 PL=0
MOVL C01026 V=800.0 PL=0
MOVL C01027 V=800.0 PL=0
MOVL C01028 V=800.0 PL=0
MOVL C01029 V=800.0 PL=0
MOVL C01030 V=800.0 PL=0
MOVL C01031 V=800.0 PL=0
MOVL C01032 V=800.0 PL=0
MOVL C01033 V=800.0 PL=0
MOVL C01034 V=800.0 PL=0
MOVL C01035 V=800.0 PL=0
MOVL C01036 V=800.0 PL=0
MOVL C01037 V=800.0 PL=0
MOVL C01038 V=800.0 PL=0
MOVL C01039 V=800.0 PL=0
MOVL C01040 V=800.0 PL=0
MOVL C01041 V=800.0 PL=0
MOVL C01042 V=800.0 PL=0
MOVL C01043 V=800.0 PL=0
MOVL C01044 V=800.0 PL=0
MOVL C01045 V=800.0 PL=0
MOVL C01046 V=800.0 PL=0
MOVL C01047 V=800.0 PL=0
MOVL C01048 V=800.0 PL=0
MOVL C01049 V=800.0 PL=0
MOVL C01050 V=800.0 PL=0
MOVL C01051 V=800.0 PL=0
MOVL C01052 V=800.0 PL=0
MOVL C01053 V=800.0 PL=0
MOVL C01054 V=800.0 PL=0
MOVL C01055 V=800.0 PL=0
MOVL C01056 V=800.0 PL=0
MOVL C01057 V=800.0 PL=0
MOVL C01058 V=800.0 PL=0
MOVL C01059 V=800.0 PL=0
MOVL C01060 V=800.0 PL=0
MOVL C01061 V=800.0 PL=0
MOVL C01062 V=800.0 PL=0
MOVL C01063 V=800.0 PL=0
MOVL C01064 V=800.0 PL=0
MOVL C01065 V=800.0 PL=0
MOVL C01066 V=800.0 PL=0
MOVL C01067 V=800.0 PL=0
MOVL C01068 V=800.0 PL=0
MOVL C01069 V=800.0 PL=0
MOVL C01070 V=800.0 PL=0
MOVL C01071 V=800.0 PL=0
MOVL C01072 V=800.0 PL=0
MOVL C01073 V=800.0 PL=0
MOVL C01074 V=800.0 PL=0
MOVL C01075 V=800.0 PL=0
MOVL C01076 V=800.0 PL=0
MOVL C01077 V=800.0 PL=0
MOVL C01078 V=800.0 PL=0
MOVL C01079 V=800.0 PL=0
MOVL C01080 V=800.0 PL=0
MOVL C01081 V=800.0 PL=0
MOVL C01082 V=800.0 PL=0
MOVL C01083 V=800.0 PL=0
MOVL C01084 V=800.0 PL=0
MOVL C01085 V=800.0 PL=0
MOVL C01086 V=800.0 PL=0
MOVL C01087 V=800.0 PL=0
MOVL C01088 V=800.0 PL=0
MOVL C01089 V=800.0 PL=0
MOVL C01090 V=800.0 PL=0
MOVL C01091 V=800.0 PL=0
MOVL C01092 V=800.0 PL=0
MOVL C01093 V=800.0 PL=0
MOVL C01094 V=800.0 PL=0
MOVL C01095 V=800.0 PL=0
MOVL C01096 V=800.0 PL=0
MOVL C01097 V=800.0 PL=0
MOVL C01098 V=800.0 PL=0
MOVL C01099 V=800.0 PL=0
MOVL C01100 V=800.0 PL=0
MOVL C01101 V=800.0 PL=0
MOVL C01102 V=800.0 PL=0
MOVL C01103 V=800.0 PL=0
MOVL C01104 V=800.0 PL=0
MOVL C01105 V=800.0 PL=0
MOVL C01106 V=800.0 PL=0
MOVL C01107 V=800.0 PL=0
MOVL C01108 V=800.0 PL=0
MOVL C01109 V=800.0 PL=0
MOVL C01110 V=800.0 PL=0
MOVL C01111 V=800.0 PL=0
MOVL C01112 V=800.0 PL=0
MOVL C01113 V=800.0 PL=0
MOVL C01114 V=800.0 PL=0
MOVL C01115 V=800.0 PL=0
MOVL C01116 V=800.0 PL=0
MOVL C01117 V=800.0 PL=0
MOVL C01118 V=800.0 PL=0
MOVL C01119 V=800.0 PL=0
MOVL C01120 V=800.0 PL=0
MOVL C01121 V=800.0 PL=0
MOVL C01122 V=800.0 PL=0
MOVL C01123 V=800.0 PL=0
MOVL C01124 V=800.0 PL=0
MOVL C01125 V=800.0 PL=0
MOVL C01126 V=800.0 PL=0
MOVL C01127 V=800.0 PL=0
MOVL C01128 V=800.0 PL=0
MOVL C01129 V=800.0 PL=0
MOVL C01130 V=800.0 PL=0
MOVL C01131 V=800.0 PL=0
MOVL C01132 V=800.0 PL=0
MOVL C01133 V=800.0 PL=0
MOVL C01134 V=800.0 PL=0
MOVL C01135 V=800.0 PL=0
MOVL C01136 V=800.0 PL=0
MOVL C01137 V=800.0 PL=0
MOVL C01138 V=800.0 PL=0
MOVL C01139 V=800.0 PL=0
MOVL C01140 V=800.0 PL=0
MOVL C01141 V=800.0 PL=0
MOVL C01142 V=800.0 PL=0
MOVL C01143 V=800.0 PL=0
MOVL C01144 V=800.0 PL=0
MOVL C01145 V=800.0 PL=0
MOVL C01146 V=800.0 PL=0
MOVL C01147 V=800.0 PL=0
MOVL C01148 V=800.0 PL=0
MOVL C01149 V=800.0 PL=0
MOVL C01150 V=800.0 PL=0
MOVL C01151 V=800.0 PL=0
MOVL C01152 V=800.0 PL=0
MOVL C01153 V=800.0 PL=0
MOVL C01154 V=800.0 PL=0
MOVL C01155 V=800.0 PL=0
MOVL C01156 V=800.0 PL=0
MOVL C01157 V=800.0 PL=0
MOVL C01158 V=800.0 PL=0
MOVL C01159 V=800.0 PL=0
MOVL C01160 V=800.0 PL=0
MOVL C01161 V=800.0 PL=0
MOVL C01162 V=800.0 PL=0
MOVL C01163 V=800.0 PL=0
MOVL C01164 V=800.0 PL=0
MOVL C01165 V=800.0 PL=0
MOVL C01166 V=800.0 PL=0
MOVL C01167 V=800.0 PL=0
MOVL C01168 V=800.0 PL=0
MOVL C01169 V=800.0 PL=0
MOVL C01170 V=800.0 PL=0
MOVL C01171 V=800.0 PL=0
MOVL C01172 V=800.0 PL=0
MOVL C01173 V=800.0 PL=0
MOVL C01174 V=800.0 PL=0
MOVL C01175 V=800.0 PL=0
MOVL C01176 V=800.0 PL=0
MOVL C01177 V=800.0 PL=0
MOVL C01178 V=800.0 PL=0
MOVL C01179 V=800.0 PL=0
MOVL C01180 V=800.0 PL=0
MOVL C01181 V=800.0 PL=0
MOVL C01182 V=800.0 PL=0
MOVL C01183 V=800.0 PL=0
MOVL C01184 V=800.0 PL=0
MOVL C01185 V=800.0 PL=0
MOVL C01186 V=800.0 PL=0
MOVL C01187 V=800.0 PL=0
MOVL C01188 V=800.0 PL=0
MOVL C01189 V=800.0 PL=0
MOVL C01190 V=800.0 PL=0
MOVL C01191 V=800.0 PL=0
MOVL C01192 V=800.0 PL=0
MOVL C01193 V=800.0 PL=0
MOVL C01194 V=800.0 PL=0
MOVL C01195 V=800.0 PL=0
MOVL C01196 V=800.0 PL=0
MOVL C01197 V=800.0 PL=0
MOVL C01198 V=800.0 PL=0
MOVL C01199 V=800.0 PL=0
MOVL C01200 V=800.0 PL=0
MOVL C01201 V=800.0 PL=0
MOVL C01202 V=800.0 PL=0
MOVL C01203 V=800.0 PL=0
MOVL C01204 V=800.0 PL=0
MOVL C01205 V=800.0 PL=0
MOVL C01206 V=800.0 PL=0
MOVL C01207 V=800.0 PL=0
MOVL C01208 V=800.0 PL=0
MOVL C01209 V=800.0 PL=0
MOVL C01210 V=800.0 PL=0
MOVL C01211 V=800.0 PL=0
MOVL C01212 V=800.0 PL=0
MOVL C01213 V=800.0 PL=0
MOVL C01214 V=800.0 PL=0
MOVL C01215 V=800.0 PL=0
MOVL C01216 V=800.0 PL=0
MOVL C01217 V=800.0 PL=0
MOVL C01218 V=800.0 PL=0
MOVL C01219 V=800.0 PL=0
MOVL C01220 V=800.0 PL=0
MOVL C01221 V=800.0 PL=0
MOVL C01222 V=800.0 PL=0
MOVL C01223 V=800.0 PL=0
MOVL C01224 V=800.0 PL=0
MOVL C01225 V=800.0 PL=0
MOVL C01226 V=800.0 PL=0
MOVL C01227 V=800.0 PL=0
MOVL C01228 V=800.0 PL=0
MOVL C01229 V=800.0 PL=0
MOVL C01230 V=800.0 PL=0
MOVL C01231 V=800.0 PL=0
MOVL C01232 V=800.0 PL=0
MOVL C01233 V=800.0 PL=0
MOVL C01234 V=800.0 PL=0
MOVL C01235 V=800.0 PL=0
MOVL C01236 V=800.0 PL=0
MOVL C01237 V=800.0 PL=0
MOVL C01238 V=800.0 PL=0
MOVL C01239 V=800.0 PL=0
MOVL C01240 V=800.0 PL=0
MOVL C01241 V=800.0 PL=0
MOVL C01242 V=800.0 PL=0
MOVL C01243 V=800.0 PL=0
MOVL C01244 V=800.0 PL=0
MOVL C01245 V=800.0 PL=0
MOVL C01246 V=800.0 PL=0
MOVL C01247 V=800.0 PL=0
MOVL C01248 V=800.0 PL=0
MOVL C01249 V=800.0 PL=0
MOVL C01250 V=800.0 PL=0
MOVL C01251 V=800.0 PL=0
MOVL C01252 V=800.0 PL=0
MOVL C01253 V=800.0 PL=0
MOVL C01254 V=800.0 PL=0
MOVL C01255 V=800.0 PL=0
MOVL C01256 V=800.0 PL=0
MOVL C01257 V=800.0 PL=0
MOVL C01258 V=800.0 PL=0
MOVL C01259 V=800.0 PL=0
MOVL C01260 V=800.0 PL=0
MOVL C01261 V=800.0 PL=0
MOVL C01262 V=800.0 PL=0
MOVL C01263 V=800.0 PL=0
MOVL C01264 V=800.0 PL=0
MOVL C01265 V=800.0 PL=0
MOVL C01266 V=800.0 PL=0
MOVL C01267 V=800.0 PL=0
MOVL C01268 V=800.0 PL=0
MOVL C01269 V=800.0 PL=0
MOVL C01270 V=800.0 PL=0
MOVL C01271 V=800.0 PL=0
MOVL C01272 V=800.0 PL=0
MOVL C01273 V=800.0 PL=0
MOVL C01274 V=800.0 PL=0
MOVL C01275 V=800.0 PL=0
MOVL C01276 V=800.0 PL=0
MOVL C01277 V=800.0 PL=0
MOVL C01278 V=800.0 PL=0
MOVL C01279 V=800.0 PL=0
MOVL C01280 V=800.0 PL=0
MOVL C01281 V=800.0 PL=0
MOVL C01282 V=800.0 PL=0
MOVL C01283 V=800.0 PL=0
MOVL C01284 V=800.0 PL=0
MOVL C01285 V=800.0 PL=0
MOVL C01286 V=800.0 PL=0
MOVL C01287 V=800.0 PL=0
MOVL C01288 V=800.0 PL=0
MOVL C01289 V=800.0 PL=0
MOVL C01290 V=800.0 PL=0
MOVL C01291 V=800.0 PL=0
MOVL C01292 V=800.0 PL=0
MOVL C01293 V=800.0 PL=0
MOVL C01294 V=800.0 PL=0
MOVL C01295 V=800.0 PL=0
MOVL C01296 V=800.0 PL=0
MOVL C01297 V=800.0 PL=0
MOVL C01298 V=800.0 PL=0
MOVL C01299 V=800.0 PL=0
MOVL C01300 V=800.0 PL=0
MOVL C01301 V=800.0 PL=0
MOVL C01302 V=800.0 PL=0
MOVL C01303 V=800.0 PL=0
MOVL C01304 V=800.0 PL=0
MOVL C01305 V=800.0 PL=0
MOVL C01306 V=800.0 PL=0
MOVL C01307 V=800.0 PL=0
MOVL C01308 V=800.0 PL=0
MOVL C01309 V=800.0 PL=0
MOVL C01310 V=800.0 PL=0
MOVL C01311 V=800.0 PL=0
MOVL C01312 V=800.0 PL=0
MOVL C01313 V=800.0 PL=0
MOVL C01314 V=800.0 PL=0
MOVL C01315 V=800.0 PL=0
MOVL C01316 V=800.0 PL=0
MOVL C01317 V=800.0 PL=0
MOVL C01318 V=800.0 PL=0
MOVL C01319 V=800.0 PL=0
MOVL C01320 V=800.0 PL=0
MOVL C01321 V=800.0 PL=0
MOVL C01322 V=800.0 PL=0
MOVL C01323 V=800.0 PL=0
MOVL C01324 V=800.0 PL=0
MOVL C01325 V=800.0 PL=0
MOVL C01326 V=800.0 PL=0
MOVL C01327 V=800.0 PL=0
MOVL C01328 V=800.0 PL=0
MOVL C01329 V=800.0 PL=0
MOVL C01330 V=800.0 PL=0
MOVL C01331 V=800.0 PL=0
MOVL C01332 V=800.0 PL=0
MOVL C01333 V=800.0 PL=0
MOVL C01334 V=800.0 PL=0
MOVL C01335 V=800.0 PL=0
MOVL C01336 V=800.0 PL=0
MOVL C01337 V=800.0 PL=0
MOVL C01338 V=800.0 PL=0
MOVL C01339 V=800.0 PL=0
MOVL C01340 V=800.0 PL=0
MOVL C01341 V=800.0 PL=0
MOVL C01342 V=800.0 PL=0
MOVL C01343 V=800.0 PL=0
MOVL C01344 V=800.0 PL=0
MOVL C01345 V=800.0 PL=0
MOVL C01346 V=800.0 PL=0
MOVL C01347 V=800.0 PL=0
MOVL C01348 V=800.0 PL=0
MOVL C01349 V=800.0 PL=0
MOVL C01350 V=800.0 PL=0
MOVL C01351 V=800.0 PL=0
MOVL C01352 V=800.0 PL=0
MOVL C01353 V=800.0 PL=0
MOVL C01354 V=800.0 PL=0
MOVL C01355 V=800.0 PL=0
MOVL C01356 V=800.0 PL=0
MOVL C01357 V=800.0 PL=0
MOVL C01358 V=800.0 PL=0
MOVL C01359 V=800.0 PL=0
MOVL C01360 V=800.0 PL=0
MOVL C01361 V=800.0 PL=0
MOVL C01362 V=800.0 PL=0
MOVL C01363 V=800.0 PL=0
MOVL C01364 V=800.0 PL=0
MOVL C01365 V=800.0 PL=0
MOVL C01366 V=800.0 PL=0
MOVL C01367 V=800.0 PL=0
MOVL C01368 V=800.0 PL=0
MOVL C01369 V=800.0 PL=0
MOVL C01370 V=800.0 PL=0
MOVL C01371 V=800.0 PL=0
MOVL C01372 V=800.0 PL=0
MOVL C01373 V=800.0 PL=0
MOVL C01374 V=800.0 PL=0
MOVL C01375 V=800.0 PL=0
MOVL C01376 V=800.0 PL=0
MOVL C01377 V=800.0 PL=0
MOVL C01378 V=800.0 PL=0
MOVL C01379 V=800.0 PL=0
MOVL C01380 V=800.0 PL=0
MOVL C01381 V=800.0 PL=0
MOVL C01382 V=800.0 PL=0
MOVL C01383 V=800.0 PL=0
MOVL C01384 V=800.0 PL=0
MOVL C01385 V=800.0 PL=0
MOVL C01386 V=800.0 PL=0
MOVL C01387 V=800.0 PL=0
MOVL C01388 V=800.0 PL=0
MOVL C01389 V=800.0 PL=0
MOVL C01390 V=800.0 PL=0
MOVL C01391 V=800.0 PL=0
MOVL C01392 V=800.0 PL=0
MOVL C01393 V=800.0 PL=0
MOVL C01394 V=800.0 PL=0
MOVL C01395 V=800.0 PL=0
MOVL C01396 V=800.0 PL=0
MOVL C01397 V=800.0 PL=0
MOVL C01398 V=800.0 PL=0
MOVL C01399 V=800.0 PL=0
MOVL C01400 V=800.0 PL=0
MOVL C01401 V=800.0 PL=0
MOVL C01402 V=800.0 PL=0
MOVL C01403 V=800.0 PL=0
MOVL C01404 V=800.0 PL=0
MOVL C01405 V=800.0 PL=0
MOVL C01406 V=800.0 PL=0
MOVL C01407 V=800.0 PL=0
MOVL C01408 V=800.0 PL=0
MOVL C01409 V=800.0 PL=0
MOVL C01410 V=800.0 PL=0
MOVL C01411 V=800.0 PL=0
MOVL C01412 V=800.0 PL=0
MOVL C01413 V=800.0 PL=0
MOVL C01414 V=800.0 PL=0
MOVL C01415 V=800.0 PL=0
MOVL C01416 V=800.0 PL=0
MOVL C01417 V=800.0 PL=0
MOVL C01418 V=800.0 PL=0
MOVL C01419 V=800.0 PL=0
MOVL C01420 V=800.0 PL=0
MOVL C01421 V=800.0 PL=0
MOVL C01422 V=800.0 PL=0
MOVL C01423 V=800.0 PL=0
MOVL C01424 V=800.0 PL=0
MOVL C01425 V=800.0 PL=0
MOVL C01426 V=800.0 PL=0
MOVL C01427 V=800.0 PL=0
MOVL C01428 V=800.0 PL=0
MOVL C01429 V=800.0 PL=0
MOVL C01430 V=800.0 PL=0
MOVL C01431 V=800.0 PL=0
MOVL C01432 V=800.0 PL=0
MOVL C01433 V=800.0 PL=0
MOVL C01434 V=800.0 PL=0
MOVL C01435 V=800.0 PL=0
MOVL C01436 V=800.0 PL=0
MOVL C01437 V=800.0 PL=0
MOVL C01438 V=800.0 PL=0
MOVL C01439 V=800.0 PL=0
MOVL C01440 V=800.0 PL=0
MOVL C01441 V=800.0 PL=0
MOVL C01442 V=800.0 PL=0
MOVL C01443 V=800.0 PL=0
MOVL C01444 V=800.0 PL=0
MOVL C01445 V=800.0 PL=0
MOVL C01446 V=800.0 PL=0
MOVL C01447 V=800.0 PL=0
MOVL C01448 V=800.0 PL=0
MOVL C01449 V=800.0 PL=0
MOVL C01450 V=800.0 PL=0
MOVL C01451 V=800.0 PL=0
MOVL C01452 V=800.0 PL=0
MOVL C01453 V=800.0 PL=0
MOVL C01454 V=800.0 PL=0
MOVL C01455 V=800.0 PL=0
MOVL C01456 V=800.0 PL=0
MOVL C01457 V=800.0 PL=0
MOVL C01458 V=800.0 PL=0
MOVL C01459 V=800.0 PL=0
MOVL C01460 V=800.0 PL=0
MOVL C01461 V=800.0 PL=0
MOVL C01462 V=800.0 PL=0
MOVL C01463 V=800.0 PL=0
MOVL C01464 V=800.0 PL=0
MOVL C01465 V=800.0 PL=0
MOVL C01466 V=800.0 PL=0
MOVL C01467 V=800.0 PL=0
MOVL C01468 V=800.0 PL=0
MOVL C01469 V=800.0 PL=0
MOVL C01470 V=800.0 PL=0
MOVL C01471 V=800.0 PL=0
MOVL C01472 V=800.0 PL=0
MOVL C01473 V=800.0 PL=0
MOVL C01474 V=800.0 PL=0
MOVL C01475 V=800.0 PL=0
MOVL C01476 V=800.0 PL=0
MOVL C01477 V=800.0 PL=0
MOVL C01478 V=800.0 PL=0
MOVL C01479 V=800.0 PL=0
MOVL C01480 V=800.0 PL=0
MOVL C01481 V=800.0 PL=0
MOVL C01482 V=800.0 PL=0
MOVL C01483 V=800.0 PL=0
MOVL C01484 V=800.0 PL=0
MOVL C01485 V=800.0 PL=0
MOVL C01486 V=800.0 PL=0
MOVL C01487 V=800.0 PL=0
MOVL C01488 V=800.0 PL=0
MOVL C01489 V=800.0 PL=0
MOVL C01490 V=800.0 PL=0
MOVL C01491 V=800.0 PL=0
MOVL C01492 V=800.0 PL=0
MOVL C01493 V=800.0 PL=0
MOVL C01494 V=800.0 PL=0
MOVL C01495 V=800.0 PL=0
MOVL C01496 V=800.0 PL=0
MOVL C01497 V=800.0 PL=0
MOVL C01498 V=800.0 PL=0
MOVL C01499 V=800.0 PL=0
MOVL C01500 V=800.0 PL=0
MOVL C01501 V=800.0 PL=0
MOVL C01502 V=800.0 PL=0
MOVL C01503 V=800.0 PL=0
MOVL C01504 V=800.0 PL=0
MOVL C01505 V=800.0 PL=0
MOVL C01506 V=800.0 PL=0
MOVL C01507 V=800.0 PL=0
MOVL C01508 V=800.0 PL=0
MOVL C01509 V=800.0 PL=0
MOVL C01510 V=800.0 PL=0
MOVL C01511 V=800.0 PL=0
MOVL C01512 V=800.0 PL=0
MOVL C01513 V=800.0 PL=0
MOVL C01514 V=800.0 PL=0
MOVL C01515 V=800.0 PL=0
MOVL C01516 V=800.0 PL=0
MOVL C01517 V=800.0 PL=0
MOVL C01518 V=800.0 PL=0
MOVL C01519 V=800.0 PL=0
MOVL C01520 V=800.0 PL=0
MOVL C01521 V=800.0 PL=0
MOVL C01522 V=800.0 PL=0
MOVL C01523 V=800.0 PL=0
MOVL C01524 V=800.0 PL=0
MOVL C01525 V=800.0 PL=0
MOVL C01526 V=800.0 PL=0
MOVL C01527 V=800.0 PL=0
MOVL C01528 V=800.0 PL=0
MOVL C01529 V=800.0 PL=0
MOVL C01530 V=800.0 PL=0
MOVL C01531 V=800.0 PL=0
MOVL C01532 V=800.0 PL=0
MOVL C01533 V=800.0 PL=0
MOVL C01534 V=800.0 PL=0
MOVL C01535 V=800.0 PL=0
MOVL C01536 V=800.0 PL=0
MOVL C01537 V=800.0 PL=0
MOVL C01538 V=800.0 PL=0
MOVL C01539 V=800.0 PL=0
MOVL C01540 V=800.0 PL=0
MOVL C01541 V=800.0 PL=0
MOVL C01542 V=800.0 PL=0
MOVL C01543 V=800.0 PL=0
MOVL C01544 V=800.0 PL=0
MOVL C01545 V=800.0 PL=0
MOVL C01546 V=800.0 PL=0
MOVL C01547 V=800.0 PL=0
MOVL C01548 V=800.0 PL=0
MOVL C01549 V=800.0 PL=0
MOVL C01550 V=800.0 PL=0
MOVL C01551 V=800.0 PL=0
MOVL C01552 V=800.0 PL=0
MOVL C01553 V=800.0 PL=0
MOVL C01554 V=800.0 PL=0
MOVL C01555 V=800.0 PL=0
MOVL C01556 V=800.0 PL=0
MOVL C01557 V=800.0 PL=0
MOVL C01558 V=800.0 PL=0
MOVL C01559 V=800.0 PL=0
MOVL C01560 V=800.0 PL=0
MOVL C01561 V=800.0 PL=0
MOVL C01562 V=800.0 PL=0
MOVL C01563 V=800.0 PL=0
MOVL C01564 V=800.0 PL=0
MOVL C01565 V=800.0 PL=0
MOVL C01566 V=800.0 PL=0
MOVL C01567 V=800.0 PL=0
MOVL C01568 V=800.0 PL=0
MOVL C01569 V=800.0 PL=0
MOVL C01570 V=800.0 PL=0
MOVL C01571 V=800.0 PL=0
MOVL C01572 V=800.0 PL=0
MOVL C01573 V=800.0 PL=0
MOVL C01574 V=800.0 PL=0
MOVL C01575 V=800.0 PL=0
MOVL C01576 V=800.0 PL=0
MOVL C01577 V=800.0 PL=0
MOVL C01578 V=800.0 PL=0
MOVL C01579 V=800.0 PL=0
MOVL C01580 V=800.0 PL=0
MOVL C01581 V=800.0 PL=0
MOVL C01582 V=800.0 PL=0
MOVL C01583 V=800.0 PL=0
MOVL C01584 V=800.0 PL=0
MOVL C01585 V=800.0 PL=0
MOVL C01586 V=800.0 PL=0
MOVL C01587 V=800.0 PL=0
MOVL C01588 V=800.0 PL=0
MOVL C01589 V=800.0 PL=0
MOVL C01590 V=800.0 PL=0
MOVL C01591 V=800.0 PL=0
MOVL C01592 V=800.0 PL=0
MOVL C01593 V=800.0 PL=0
MOVL C01594 V=800.0 PL=0
MOVL C01595 V=800.0 PL=0
MOVL C01596 V=800.0 PL=0
MOVL C01597 V=800.0 PL=0
MOVL C01598 V=800.0 PL=0
MOVL C01599 V=800.0 PL=0
MOVL C01600 V=800.0 PL=0
MOVL C01601 V=800.0 PL=0
MOVL C01602 V=800.0 PL=0
MOVL C01603 V=800.0 PL=0
MOVL C01604 V=800.0 PL=0
MOVL C01605 V=800.0 PL=0
MOVL C01606 V=800.0 PL=0
MOVL C01607 V=800.0 PL=0
MOVL C01608 V=800.0 PL=0
MOVL C01609 V=800.0 PL=0
MOVL C01610 V=800.0 PL=0
MOVL C01611 V=800.0 PL=0
MOVL C01612 V=800.0 PL=0
MOVL C01613 V=800.0 PL=0
MOVL C01614 V=800.0 PL=0
MOVL C01615 V=800.0 PL=0
MOVL C01616 V=800.0 PL=0
MOVL C01617 V=800.0 PL=0
MOVL C01618 V=800.0 PL=0
MOVL C01619 V=800.0 PL=0
MOVL C01620 V=800.0 PL=0
MOVL C01621 V=800.0 PL=0
MOVL C01622 V=800.0 PL=0
MOVL C01623 V=800.0 PL=0
MOVL C01624 V=800.0 PL=0
MOVL C01625 V=800.0 PL=0
MOVL C01626 V=800.0 PL=0
MOVL C01627 V=800.0 PL=0
MOVL C01628 V=800.0 PL=0
MOVL C01629 V=800.0 PL=0
MOVL C01630 V=800.0 PL=0
MOVL C01631 V=800.0 PL=0
MOVL C01632 V=800.0 PL=0
MOVL C01633 V=800.0 PL=0
MOVL C01634 V=800.0 PL=0
MOVL C01635 V=800.0 PL=0
MOVL C01636 V=800.0 PL=0
MOVL C01637 V=800.0 PL=0
MOVL C01638 V=800.0 PL=0
MOVL C01639 V=800.0 PL=0
MOVL C01640 V=800.0 PL=0
MOVL C01641 V=800.0 PL=0
MOVL C01642 V=800.0 PL=0
MOVL C01643 V=800.0 PL=0
MOVL C01644 V=800.0 PL=0
MOVL C01645 V=800.0 PL=0
MOVL C01646 V=800.0 PL=0
MOVL C01647 V=800.0 PL=0
MOVL C01648 V=800.0 PL=0
MOVL C01649 V=800.0 PL=0
MOVL C01650 V=800.0 PL=0
MOVL C01651 V=800.0 PL=0
MOVL C01652 V=800.0 PL=0
MOVL C01653 V=800.0 PL=0
MOVL C01654 V=800.0 PL=0
MOVL C01655 V=800.0 PL=0
MOVL C01656 V=800.0 PL=0
MOVL C01657 V=800.0 PL=0
MOVL C01658 V=800.0 PL=0
MOVL C01659 V=800.0 PL=0
MOVL C01660 V=800.0 PL=0
MOVL C01661 V=800.0 PL=0
MOVL C01662 V=800.0 PL=0
MOVL C01663 V=800.0 PL=0
MOVL C01664 V=800.0 PL=0
MOVL C01665 V=800.0 PL=0
MOVL C01666 V=800.0 PL=0
MOVL C01667 V=800.0 PL=0
MOVL C01668 V=800.0 PL=0
MOVL C01669 V=800.0 PL=0
MOVL C01670 V=800.0 PL=0
MOVL C01671 V=800.0 PL=0
MOVL C01672 V=800.0 PL=0
MOVL C01673 V=800.0 PL=0
MOVL C01674 V=800.0 PL=0
MOVL C01675 V=800.0 PL=0
MOVL C01676 V=800.0 PL=0
MOVL C01677 V=800.0 PL=0
MOVL C01678 V=800.0 PL=0
MOVL C01679 V=800.0 PL=0
MOVL C01680 V=800.0 PL=0
MOVL C01681 V=800.0 PL=0
MOVL C01682 V=800.0 PL=0
MOVL C01683 V=800.0 PL=0
MOVL C01684 V=800.0 PL=0
MOVL C01685 V=800.0 PL=0
MOVL C01686 V=800.0 PL=0
MOVL C01687 V=800.0 PL=0
MOVL C01688 V=800.0 PL=0
MOVL C01689 V=800.0 PL=0
MOVL C01690 V=800.0 PL=0
MOVL C01691 V=800.0 PL=0
MOVL C01692 V=800.0 PL=0
MOVL C01693 V=800.0 PL=0
MOVL C01694 V=800.0 PL=0
MOVL C01695 V=800.0 PL=0
MOVL C01696 V=800.0 PL=0
MOVL C01697 V=800.0 PL=0
MOVL C01698 V=800.0 PL=0
MOVL C01699 V=800.0 PL=0
MOVL C01700 V=800.0 PL=0
MOVL C01701 V=800.0 PL=0
MOVL C01702 V=800.0 PL=0
MOVL C01703 V=800.0 PL=0
MOVL C01704 V=800.0 PL=0
MOVL C01705 V=800.0 PL=0
MOVL C01706 V=800.0 PL=0
MOVL C01707 V=800.0 PL=0
MOVL C01708 V=800.0 PL=0
MOVL C01709 V=800.0 PL=0
MOVL C01710 V=800.0 PL=0
MOVL C01711 V=800.0 PL=0
MOVL C01712 V=800.0 PL=0
MOVL C01713 V=800.0 PL=0
MOVL C01714 V=800.0 PL=0
MOVL C01715 V=800.0 PL=0
MOVL C01716 V=800.0 PL=0
MOVL C01717 V=800.0 PL=0
MOVL C01718 V=800.0 PL=0
MOVL C01719 V=800.0 PL=0
MOVL C01720 V=800.0 PL=0
MOVL C01721 V=800.0 PL=0
MOVL C01722 V=800.0 PL=0
MOVL C01723 V=800.0 PL=0
MOVL C01724 V=800.0 PL=0
MOVL C01725 V=800.0 PL=0
MOVL C01726 V=800.0 PL=0
MOVL C01727 V=800.0 PL=0
MOVL C01728 V=800.0 PL=0
MOVL C01729 V=800.0 PL=0
MOVL C01730 V=800.0 PL=0
MOVL C01731 V=800.0 PL=0
MOVL C01732 V=800.0 PL=0
MOVL C01733 V=800.0 PL=0
MOVL C01734 V=800.0 PL=0
MOVL C01735 V=800.0 PL=0
MOVL C01736 V=800.0 PL=0
MOVL C01737 V=800.0 PL=0
MOVL C01738 V=800.0 PL=0
MOVL C01739 V=800.0 PL=0
MOVL C01740 V=800.0 PL=0
MOVL C01741 V=800.0 PL=0
MOVL C01742 V=800.0 PL=0
MOVL C01743 V=800.0 PL=0
MOVL C01744 V=800.0 PL=0
MOVL C01745 V=800.0 PL=0
MOVL C01746 V=800.0 PL=0
MOVL C01747 V=800.0 PL=0
MOVL C01748 V=800.0 PL=0
MOVL C01749 V=800.0 PL=0
MOVL C01750 V=800.0 PL=0
MOVL C01751 V=800.0 PL=0
MOVL C01752 V=800.0 PL=0
MOVL C01753 V=800.0 PL=0
MOVL C01754 V=800.0 PL=0
MOVL C01755 V=800.0 PL=0
MOVL C01756 V=800.0 PL=0
MOVL C01757 V=800.0 PL=0
MOVL C01758 V=800.0 PL=0
MOVL C01759 V=800.0 PL=0
MOVL C01760 V=800.0 PL=0
MOVL C01761 V=800.0 PL=0
MOVL C01762 V=800.0 PL=0
MOVL C01763 V=800.0 PL=0
MOVL C01764 V=800.0 PL=0
MOVL C01765 V=800.0 PL=0
MOVL C01766 V=800.0 PL=0
MOVL C01767 V=800.0 PL=0
MOVL C01768 V=800.0 PL=0
MOVL C01769 V=800.0 PL=0
MOVL C01770 V=800.0 PL=0
MOVL C01771 V=800.0 PL=0
MOVL C01772 V=800.0 PL=0
MOVL C01773 V=800.0 PL=0
MOVL C01774 V=800.0 PL=0
MOVL C01775 V=800.0 PL=0
MOVL C01776 V=800.0 PL=0
MOVL C01777 V=800.0 PL=0
MOVL C01778 V=800.0 PL=0
MOVL C01779 V=800.0 PL=0
MOVL C01780 V=800.0 PL=0
MOVL C01781 V=800.0 PL=0
MOVL C01782 V=800.0 PL=0
MOVL C01783 V=800.0 PL=0
MOVL C01784 V=800.0 PL=0
MOVL C01785 V=800.0 PL=0
MOVL C01786 V=800.0 PL=0
MOVL C01787 V=800.0 PL=0
MOVL C01788 V=800.0 PL=0
MOVL C01789 V=800.0 PL=0
MOVL C01790 V=800.0 PL=0
MOVL C01791 V=800.0 PL=0
MOVL C01792 V=800.0 PL=0
MOVL C01793 V=800.0 PL=0
MOVL C01794 V=800.0 PL=0
MOVL C01795 V=800.0 PL=0
MOVL C01796 V=800.0 PL=0
MOVL C01797 V=800.0 PL=0
MOVL C01798 V=800.0 PL=0
MOVL C01799 V=800.0 PL=0
MOVL C01800 V=800.0 PL=0
MOVL C01801 V=800.0 PL=0
MOVL C01802 V=800.0 PL=0
MOVL C01803 V=800.0 PL=0
MOVL C01804 V=800.0 PL=0
MOVL C01805 V=800.0 PL=0
MOVL C01806 V=800.0 PL=0
MOVL C01807 V=800.0 PL=0
MOVL C01808 V=800.0 PL=0
MOVL C01809 V=800.0 PL=0
MOVL C01810 V=800.0 PL=0
MOVL C01811 V=800.0 PL=0
MOVL C01812 V=800.0 PL=0
MOVL C01813 V=800.0 PL=0
MOVL C01814 V=800.0 PL=0
MOVL C01815 V=800.0 PL=0
MOVL C01816 V=800.0 PL=0
MOVL C01817 V=800.0 PL=0
MOVL C01818 V=800.0 PL=0
MOVL C01819 V=800.0 PL=0
MOVL C01820 V=800.0 PL=0
MOVL C01821 V=800.0 PL=0
MOVL C01822 V=800.0 PL=0
MOVL C01823 V=800.0 PL=0
MOVL C01824 V=800.0 PL=0
MOVL C01825 V=800.0 PL=0
MOVL C01826 V=800.0 PL=0
MOVL C01827 V=800.0 PL=0
MOVL C01828 V=800.0 PL=0
MOVL C01829 V=800.0 PL=0
MOVL C01830 V=800.0 PL=0
MOVL C01831 V=800.0 PL=0
MOVL C01832 V=800.0 PL=0
MOVL C01833 V=800.0 PL=0
MOVL C01834 V=800.0 PL=0
MOVL C01835 V=800.0 PL=0
MOVL C01836 V=800.0 PL=0
MOVL C01837 V=800.0 PL=0
MOVL C01838 V=800.0 PL=0
MOVL C01839 V=800.0 PL=0
MOVL C01840 V=800.0 PL=0
MOVL C01841 V=800.0 PL=0
MOVL C01842 V=800.0 PL=0
MOVL C01843 V=800.0 PL=0
MOVL C01844 V=800.0 PL=0
MOVL C01845 V=800.0 PL=0
MOVL C01846 V=800.0 PL=0
MOVL C01847 V=800.0 PL=0
MOVL C01848 V=800.0 PL=0
MOVL C01849 V=800.0 PL=0
MOVL C01850 V=800.0 PL=0
MOVL C01851 V=800.0 PL=0
MOVL C01852 V=800.0 PL=0
MOVL C01853 V=800.0 PL=0
MOVL C01854 V=800.0 PL=0
MOVL C01855 V=800.0 PL=0
MOVL C01856 V=800.0 PL=0
MOVL C01857 V=800.0 PL=0
MOVL C01858 V=800.0 PL=0
MOVL C01859 V=800.0 PL=0
MOVL C01860 V=800.0 PL=0
MOVL C01861 V=800.0 PL=0
MOVL C01862 V=800.0 PL=0
MOVL C01863 V=800.0 PL=0
MOVL C01864 V=800.0 PL=0
MOVL C01865 V=800.0 PL=0
MOVL C01866 V=800.0 PL=0
MOVL C01867 V=800.0 PL=0
MOVL C01868 V=800.0 PL=0
MOVL C01869 V=800.0 PL=0
MOVL C01870 V=800.0 PL=0
MOVL C01871 V=800.0 PL=0
MOVL C01872 V=800.0 PL=0
MOVL C01873 V=800.0 PL=0
MOVL C01874 V=800.0 PL=0
MOVL C01875 V=800.0 PL=0
MOVL C01876 V=800.0 PL=0
MOVL C01877 V=800.0 PL=0
MOVL C01878 V=800.0 PL=0
MOVL C01879 V=800.0 PL=0
MOVL C01880 V=800.0 PL=0
MOVL C01881 V=800.0 PL=0
MOVL C01882 V=800.0 PL=0
MOVL C01883 V=800.0 PL=0
MOVL C01884 V=800.0 PL=0
MOVL C01885 V=800.0 PL=0
MOVL C01886 V=800.0 PL=0
MOVL C01887 V=800.0 PL=0
MOVL C01888 V=800.0 PL=0
MOVL C01889 V=800.0 PL=0
MOVL C01890 V=800.0 PL=0
MOVL C01891 V=800.0 PL=0
MOVL C01892 V=800.0 PL=0
MOVL C01893 V=800.0 PL=0
MOVL C01894 V=800.0 PL=0
MOVL C01895 V=800.0 PL=0
MOVL C01896 V=800.0 PL=0
MOVL C01897 V=800.0 PL=0
MOVL C01898 V=800.0 PL=0
MOVL C01899 V=800.0 PL=0
MOVL C01900 V=800.0 PL=0
MOVL C01901 V=800.0 PL=0
MOVL C01902 V=800.0 PL=0
MOVL C01903 V=800.0 PL=0
MOVL C01904 V=800.0 PL=0
MOVL C01905 V=800.0 PL=0
MOVL C01906 V=800.0 PL=0
MOVL C01907 V=800.0 PL=0
MOVL C01908 V=800.0 PL=0
MOVL C01909 V=800.0 PL=0
MOVL C01910 V=800.0 PL=0
MOVL C01911 V=800.0 PL=0
MOVL C01912 V=800.0 PL=0
MOVL C01913 V=800.0 PL=0
MOVL C01914 V=800.0 PL=0
MOVL C01915 V=800.0 PL=0
MOVL C01916 V=800.0 PL=0
MOVL C01917 V=800.0 PL=0
MOVL C01918 V=800.0 PL=0
MOVL C01919 V=800.0 PL=0
MOVL C01920 V=800.0 PL=0
MOVL C01921 V=800.0 PL=0
MOVL C01922 V=800.0 PL=0
MOVL C01923 V=800.0 PL=0
MOVL C01924 V=800.0 PL=0
MOVL C01925 V=800.0 PL=0
MOVL C01926 V=800.0 PL=0
MOVL C01927 V=800.0 PL=0
MOVL C01928 V=800.0 PL=0
MOVL C01929 V=800.0 PL=0
MOVL C01930 V=800.0 PL=0
MOVL C01931 V=800.0 PL=0
MOVL C01932 V=800.0 PL=0
MOVL C01933 V=800.0 PL=0
MOVL C01934 V=800.0 PL=0
MOVL C01935 V=800.0 PL=0
MOVL C01936 V=800.0 PL=0
MOVL C01937 V=800.0 PL=0
MOVL C01938 V=800.0 PL=0
MOVL C01939 V=800.0 PL=0
MOVL C01940 V=800.0 PL=0
MOVL C01941 V=800.0 PL=0
MOVL C01942 V=800.0 PL=0
MOVL C01943 V=800.0 PL=0
MOVL C01944 V=800.0 PL=0
MOVL C01945 V=800.0 PL=0
MOVL C01946 V=800.0 PL=0
MOVL C01947 V=800.0 PL=0
MOVL C01948 V=800.0 PL=0
MOVL C01949 V=800.0 PL=0
MOVL C01950 V=800.0 PL=0
MOVL C01951 V=800.0 PL=0
MOVL C01952 V=800.0 PL=0
MOVL C01953 V=800.0 PL=0
MOVL C01954 V=800.0 PL=0
MOVL C01955 V=800.0 PL=0
MOVL C01956 V=800.0 PL=0
MOVL C01957 V=800.0 PL=0
MOVL C01958 V=800.0 PL=0
MOVL C01959 V=800.0 PL=0
MOVL C01960 V=800.0 PL=0
MOVL C01961 V=800.0 PL=0
MOVL C01962 V=800.0 PL=0
MOVL C01963 V=800.0 PL=0
MOVL C01964 V=800.0 PL=0
MOVL C01965 V=800.0 PL=0
MOVL C01966 V=800.0 PL=0
MOVL C01967 V=800.0 PL=0
MOVL C01968 V=800.0 PL=0
MOVL C01969 V=800.0 PL=0
MOVL C01970 V=800.0 PL=0
MOVL C01971 V=800.0 PL=0
MOVL C01972 V=800.0 PL=0
MOVL C01973 V=800.0 PL=0
MOVL C01974 V=800.0 PL=0
MOVL C01975 V=800.0 PL=0
MOVL C01976 V=800.0 PL=0
MOVL C01977 V=800.0 PL=0
MOVL C01978 V=800.0 PL=0
MOVL C01979 V=800.0 PL=0
MOVL C01980 V=800.0 PL=0
MOVL C01981 V=800.0 PL=0
MOVL C01982 V=800.0 PL=0
MOVL C01983 V=800.0 PL=0
MOVL C01984 V=800.0 PL=0
MOVL C01985 V=800.0 PL=0
MOVL C01986 V=800.0 PL=0
MOVL C01987 V=800.0 PL=0
MOVL C01988 V=800.0 PL=0
MOVL C01989 V=800.0 PL=0
MOVL C01990 V=800.0 PL=0
MOVL C01991 V=800.0 PL=0
MOVL C01992 V=800.0 PL=0
MOVL C01993 V=800.0 PL=0
MOVL C01994 V=800.0 PL=0
MOVL C01995 V=800.0 PL=0
MOVL C01996 V=800.0 PL=0
MOVL C01997 V=800.0 PL=0
